LIN {X 0,Y 187.347,Z 253.939,A -85,B 0,C 180,E1 -26155.616,E2 -26155.616} C_VEL
LIN {X 0,Y 193.474,Z 262.012,A -85,B 0,C 180,E1 -26158.88,E2 -26158.88} C_VEL
LIN {X 0,Y 201.659,Z 270.756,A -85,B 0,C 180,E1 -26162.734,E2 -26162.734} C_VEL
LIN {X 0,Y 208.52,Z 276.532,A -85,B 0,C 180,E1 -26165.504,E2 -26165.504} C_VEL
LIN {X 0,Y 219.741,Z 283.992,A -85,B 0,C 180,E1 -26169.402,E2 -26169.402} C_VEL
LIN {X 0,Y 231.619,Z 290.129,A -85,B 0,C 180,E1 -26172.899,E2 -26172.899} C_VEL
LIN {X 0,Y 242.77,Z 294.984,A -85,B 0,C 180,E1 -26175.879,E2 -26175.879} C_VEL
LIN {X 0,Y 253.839,Z 299.442,A -85,B 0,C 180,E1 -26178.825,E2 -26178.825} C_VEL
LIN {X 0,Y 260.121,Z 302.011,A -85,B 0,C 180,E1 -26180.671,E2 -26180.671} C_VEL
LIN {X 0,Y 265.393,Z 304.118,A -85,B 0,C 180,E1 -26182.391,E2 -26182.391} C_VEL
LIN {X 0,Y 269.414,Z 305.803,A -85,B 0,C 180,E1 -26184.011,E2 -26184.011} C_VEL
LIN {X 0,Y 272.285,Z 307.103,A -85,B 0,C 180,E1 -26185.559,E2 -26185.559} C_VEL
LIN {X 0,Y 274.929,Z 308.026,A -85,B 0,C 180,E1 -26187.069,E2 -26187.069} C_VEL
LIN {X 0,Y 276.549,Z 308.577,A -85,B 0,C 180,E1 -26188.544,E2 -26188.544} C_VEL
LIN {X 0,Y 277.403,Z 308.756,A -85,B 0,C 180,E1 -26190,E2 -26190} C_VEL
LIN {X 0,Y 276.553,Z 308.577,A -85,B 0,C 180,E1 -26191.456,E2 -26191.456} C_VEL
LIN {X 0,Y 274.508,Z 307.901,A -85,B 0,C 180,E1 -26193.171,E2 -26193.171} C_VEL
LIN {X 0,Y 272.281,Z 307.103,A -85,B 0,C 180,E1 -26194.441,E2 -26194.441} C_VEL
LIN {X 0,Y 268.688,Z 305.506,A -85,B 0,C 180,E1 -26196.312,E2 -26196.312} C_VEL
LIN {X 0,Y 265.387,Z 304.118,A -85,B 0,C 180,E1 -26197.609,E2 -26197.609} C_VEL
LIN {X 0,Y 260.12,Z 302.01,A -85,B 0,C 180,E1 -26199.329,E2 -26199.329} C_VEL
LIN {X 0,Y 253.786,Z 299.444,A -85,B 0,C 180,E1 -26201.177,E2 -26201.177} C_VEL
LIN {X 0,Y 242.762,Z 295.002,A -85,B 0,C 180,E1 -26204.114,E2 -26204.114} C_VEL
LIN {X 0,Y 228.839,Z 288.795,A -85,B 0,C 180,E1 -26207.885,E2 -26207.885} C_VEL
LIN {X 0,Y 218.36,Z 283.205,A -85,B 0,C 180,E1 -26211.036,E2 -26211.036} C_VEL
LIN {X 0,Y 208.502,Z 276.573,A -85,B 0,C 180,E1 -26214.485,E2 -26214.485} C_VEL
LIN {X 0,Y 199.46,Z 268.628,A -85,B 0,C 180,E1 -26218.254,E2 -26218.254} C_VEL
LIN {X 0,Y 190.254,Z 257.902,A -85,B 0,C 180,E1 -26222.823,E2 -26222.823} C_VEL
LIN {X 0,Y 183.695,Z 248.177,A -85,B 0,C 180,E1 -26226.542,E2 -26226.542} C_VEL
LIN {X 0,Y 179.378,Z 240.181,A -85,B 0,C 180,E1 -26229.305,E2 -26229.305} C_VEL
LIN {X 0,Y 174.422,Z 229.195,A -85,B 0,C 180,E1 -26232.665,E2 -26232.665} C_VEL
LIN {X 0,Y 170.348,Z 218.871,A -85,B 0,C 180,E1 -26235.465,E2 -26235.465} C_VEL
LIN {X 0,Y 166.416,Z 207.712,A -85,B 0,C 180,E1 -26238.106,E2 -26238.106} C_VEL
LIN {X 0,Y 160.97,Z 191.989,A -85,B 0,C 180,E1 -26241.487,E2 -26241.487} C_VEL
LIN {X 0,Y 157.371,Z 183.213,A -85,B 0,C 180,E1 -26243.839,E2 -26243.839} C_VEL
LIN {X 0,Y 153.272,Z 174.648,A -85,B 0,C 180,E1 -26246.72,E2 -26246.72} C_VEL
LIN {X 0,Y 148.41,Z 165.755,A -85,B 0,C 180,E1 -26250.575,E2 -26250.575} C_VEL
LIN {X 0,Y 144.141,Z 158.771,A -85,B 0,C 180,E1 -26254.555,E2 -26254.555} C_VEL
LIN {X 0,Y 141.444,Z 154.774,A -85,B 0,C 180,E1 -26257.498,E2 -26257.498} C_VEL
LIN {X 0,Y 138.938,Z 150.996,A -85,B 0,C 180,E1 -26260.746,E2 -26260.746} C_VEL
LIN {X 0,Y 136.456,Z 147.585,A -85,B 0,C 180,E1 -26264.697,E2 -26264.697} C_VEL
LIN {X 0,Y 135.796,Z 146.33,A -85,B 0,C 180,E1 -26266.035,E2 -26266.035} C_VEL
LIN {X 0,Y 133.402,Z 143.471,A -85,B 0,C 180,E1 -26272.243,E2 -26272.243} C_VEL
LIN {X 0,Y 132.743,Z 141.518,A -85,B 0,C 180,E1 -26276.207,E2 -26276.207} C_VEL
LIN {X 0,Y 132.555,Z 140.915,A -85,B 0,C 180,E1 -26280.002,E2 -26280.002} C_VEL
LIN {X 0,Y 132.834,Z 141.773,A -85,B 0,C 180,E1 -26284.174,E2 -26284.174} C_VEL
LIN {X 0,Y 135.273,Z 145.963,A -85,B 0,C 180,E1 -26292.567,E2 -26292.567} C_VEL
LIN {X 0,Y 136.019,Z 146.575,A -85,B 0,C 180,E1 -26294.018,E2 -26294.018} C_VEL
LIN {X 0,Y 138.273,Z 150.297,A -85,B 0,C 180,E1 -26297.949,E2 -26297.949} C_VEL
LIN {X 0,Y 139.397,Z 151.65,A -85,B 0,C 180,E1 -26299.514,E2 -26299.514} C_VEL
LIN {X 0,Y 142.582,Z 156.425,A -85,B 0,C 180,E1 -26303.418,E2 -26303.418} C_VEL
LIN {X 0,Y 145.517,Z 161.05,A -85,B 0,C 180,E1 -26306.44,E2 -26306.44} C_VEL
LIN {X 0,Y 147.849,Z 164.954,A -85,B 0,C 180,E1 -26308.577,E2 -26308.577} C_VEL
LIN {X 0,Y 151.514,Z 173.302,A -85,B 0,C 180,E1 -26311.749,E2 -26311.749} C_VEL
LIN {X 0,Y 155.214,Z 183.268,A -85,B 0,C 180,E1 -26314.676,E2 -26314.676} C_VEL
LIN {X 0,Y 156.563,Z 187.492,A -85,B 0,C 180,E1 -26315.703,E2 -26315.703} C_VEL
LIN {X 0,Y 154.13,Z 215.499,A -85,B 0,C 180,E1 -26316.785,E2 -26316.785} C_VEL
LIN {X 0,Y 152.014,Z 228.263,A -85,B 0,C 180,E1 -26317.567,E2 -26317.567} C_VEL
LIN {X 0,Y 148.714,Z 241.034,A -85,B 0,C 180,E1 -26318.761,E2 -26318.761} C_VEL
LIN {X 0,Y 145.534,Z 250.542,A -85,B 0,C 180,E1 -26319.949,E2 -26319.949} C_VEL
LIN {X 0,Y 141.891,Z 259.814,A -85,B 0,C 180,E1 -26321.483,E2 -26321.483} C_VEL
LIN {X 0,Y 137.763,Z 268.752,A -85,B 0,C 180,E1 -26323.368,E2 -26323.368} C_VEL
LIN {X 0,Y 133.256,Z 277.274,A -85,B 0,C 180,E1 -26325.668,E2 -26325.668} C_VEL
LIN {X 0,Y 129.044,Z 284.489,A -85,B 0,C 180,E1 -26328.152,E2 -26328.152} C_VEL
LIN {X 0,Y 125.059,Z 290.686,A -85,B 0,C 180,E1 -26330.786,E2 -26330.786} C_VEL
LIN {X 0,Y 120.616,Z 297.224,A -85,B 0,C 180,E1 -26334.361,E2 -26334.361} C_VEL
LIN {X 0,Y 115.966,Z 303.643,A -85,B 0,C 180,E1 -26338.994,E2 -26338.994} C_VEL
LIN {X 0,Y 111.959,Z 308.773,A -85,B 0,C 180,E1 -26343.934,E2 -26343.934} C_VEL
LIN {X 0,Y 108.778,Z 312.762,A -85,B 0,C 180,E1 -26349.185,E2 -26349.185} C_VEL
LIN {X 0,Y 106.69,Z 315.721,A -85,B 0,C 180,E1 -26354.723,E2 -26354.723} C_VEL
LIN {X 0,Y 105.26,Z 318.183,A -85,B 0,C 180,E1 -26362.326,E2 -26362.326} C_VEL
LIN {X 0,Y 105.046,Z 318.779,A -85,B 0,C 180,E1 -26366.164,E2 -26366.164} C_VEL
LIN {X 0,Y 105.171,Z 318.941,A -85,B 0,C 180,E1 -26370,E2 -26370} C_VEL
LIN {X 0,Y 105.039,Z 318.779,A -85,B 0,C 180,E1 -26373.836,E2 -26373.836} C_VEL
LIN {X 0,Y 105.229,Z 318.182,A -85,B 0,C 180,E1 -26377.676,E2 -26377.676} C_VEL
LIN {X 0,Y 106.69,Z 315.721,A -85,B 0,C 180,E1 -26385.277,E2 -26385.277} C_VEL
LIN {X 0,Y 108.778,Z 312.762,A -85,B 0,C 180,E1 -26390.815,E2 -26390.815} C_VEL
LIN {X 0,Y 111.96,Z 308.773,A -85,B 0,C 180,E1 -26396.066,E2 -26396.066} C_VEL
LIN {X 0,Y 115.976,Z 303.644,A -85,B 0,C 180,E1 -26401.003,E2 -26401.003} C_VEL
LIN {X 0,Y 120.658,Z 297.225,A -85,B 0,C 180,E1 -26405.625,E2 -26405.625} C_VEL
LIN {X 0,Y 126.044,Z 289.304,A -85,B 0,C 180,E1 -26409.883,E2 -26409.883} C_VEL
LIN {X 0,Y 131.143,Z 281.111,A -85,B 0,C 180,E1 -26413.1,E2 -26413.1} C_VEL
LIN {X 0,Y 136.058,Z 272.154,A -85,B 0,C 180,E1 -26415.783,E2 -26415.783} C_VEL
LIN {X 0,Y 140.108,Z 263.865,A -85,B 0,C 180,E1 -26417.721,E2 -26417.721} C_VEL
LIN {X 0,Y 144.302,Z 253.804,A -85,B 0,C 180,E1 -26419.552,E2 -26419.552} C_VEL
LIN {X 0,Y 147.751,Z 244.053,A -85,B 0,C 180,E1 -26420.889,E2 -26420.889} C_VEL
LIN {X 0,Y 150.612,Z 233.975,A -85,B 0,C 180,E1 -26421.947,E2 -26421.947} C_VEL
LIN {X 0,Y 152.841,Z 223.594,A -85,B 0,C 180,E1 -26422.756,E2 -26422.756} C_VEL
LIN {X 0,Y 154.336,Z 213.507,A -85,B 0,C 180,E1 -26423.307,E2 -26423.307} C_VEL
LIN {X 0,Y 156.557,Z 187.548,A -85,B 0,C 180,E1 -26424.295,E2 -26424.295} C_VEL
LIN {X 0,Y 153.767,Z 179.164,A -85,B 0,C 180,E1 -26426.442,E2 -26426.442} C_VEL
LIN {X 0,Y 149.574,Z 168.715,A -85,B 0,C 180,E1 -26429.888,E2 -26429.888} C_VEL
LIN {X 0,Y 146.975,Z 163.379,A -85,B 0,C 180,E1 -26432.209,E2 -26432.209} C_VEL
LIN {X 0,Y 143.653,Z 158.1,A -85,B 0,C 180,E1 -26435.426,E2 -26435.426} C_VEL
LIN {X 0,Y 141.524,Z 154.839,A -85,B 0,C 180,E1 -26437.787,E2 -26437.787} C_VEL
LIN {X 0,Y 138.836,Z 150.858,A -85,B 0,C 180,E1 -26441.267,E2 -26441.267} C_VEL
LIN {X 0,Y 138.374,Z 150.375,A -85,B 0,C 180,E1 -26441.912,E2 -26441.912} C_VEL
LIN {X 0,Y 136.784,Z 149.34,A -85,B 0,C 180,E1 -26444.241,E2 -26444.241} C_VEL
LIN {X 0,Y 134.384,Z 149.472,A -85,B 0,C 180,E1 -26448.305,E2 -26448.305} C_VEL
LIN {X 0,Y 132.917,Z 149.898,A -85,B 0,C 180,E1 -26451.671,E2 -26451.671} C_VEL
LIN {X 0,Y 132.203,Z 149.602,A -85,B 0,C 180,E1 -26454.227,E2 -26454.227} C_VEL
LIN {X 0,Y 132.052,Z 149.284,A -85,B 0,C 180,E1 -26455.075,E2 -26455.075} C_VEL
LIN {X 0,Y 131.771,Z 148.3,A -85,B 0,C 180,E1 -26457.706,E2 -26457.706} C_VEL
LIN {X 0,Y 131.686,Z 147.992,A -85,B 0,C 180,E1 -26459.998,E2 -26459.998} C_VEL
LIN {X 0,Y 131.916,Z 148.746,A -85,B 0,C 180,E1 -26464.199,E2 -26464.199} C_VEL
LIN {X 0,Y 133.989,Z 152.766,A -85,B 0,C 180,E1 -26472.109,E2 -26472.109} C_VEL
LIN {X 0,Y 134.836,Z 153.712,A -85,B 0,C 180,E1 -26473.919,E2 -26473.919} C_VEL
LIN {X 0,Y 137.218,Z 157.472,A -85,B 0,C 180,E1 -26478.163,E2 -26478.163} C_VEL
LIN {X 0,Y 140.448,Z 162.453,A -85,B 0,C 180,E1 -26482.525,E2 -26482.525} C_VEL
LIN {X 0,Y 143.306,Z 167.161,A -85,B 0,C 180,E1 -26485.702,E2 -26485.702} C_VEL
LIN {X 0,Y 146.753,Z 173.26,A -85,B 0,C 180,E1 -26489.003,E2 -26489.003} C_VEL
LIN {X 0,Y 151.229,Z 182.072,A -85,B 0,C 180,E1 -26492.72,E2 -26492.72} C_VEL
LIN {X 0,Y 155.275,Z 191.24,A -85,B 0,C 180,E1 -26495.712,E2 -26495.712} C_VEL
LIN {X 0,Y 159.125,Z 202.11,A -85,B 0,C 180,E1 -26498.394,E2 -26498.394} C_VEL
LIN {X 0,Y 163.336,Z 215.721,A -85,B 0,C 180,E1 -26501.519,E2 -26501.519} C_VEL
LIN {X 0,Y 166.6,Z 225.797,A -85,B 0,C 180,E1 -26504.181,E2 -26504.181} C_VEL
LIN {X 0,Y 170.345,Z 235.871,A -85,B 0,C 180,E1 -26507.235,E2 -26507.235} C_VEL
LIN {X 0,Y 174.011,Z 244.448,A -85,B 0,C 180,E1 -26510.117,E2 -26510.117} C_VEL
LIN {X 0,Y 178.938,Z 253.723,A -85,B 0,C 180,E1 -26513.626,E2 -26513.626} C_VEL
LIN {X 0,Y 184.314,Z 261.859,A -85,B 0,C 180,E1 -26517.019,E2 -26517.019} C_VEL
LIN {X 0,Y 190.756,Z 269.605,A -85,B 0,C 180,E1 -26520.561,E2 -26520.561} C_VEL
LIN {X 0,Y 198.398,Z 276.897,A -85,B 0,C 180,E1 -26524.191,E2 -26524.191} C_VEL
LIN {X 0,Y 208.728,Z 284.302,A -85,B 0,C 180,E1 -26528.261,E2 -26528.261} C_VEL
LIN {X 0,Y 221.275,Z 291.024,A -85,B 0,C 180,E1 -26532.33,E2 -26532.33} C_VEL
LIN {X 0,Y 235.088,Z 296.772,A -85,B 0,C 180,E1 -26536.163,E2 -26536.163} C_VEL
LIN {X 0,Y 246.761,Z 301.009,A -85,B 0,C 180,E1 -26539.289,E2 -26539.289} C_VEL
LIN {X 0,Y 255.566,Z 304.111,A -85,B 0,C 180,E1 -26541.88,E2 -26541.88} C_VEL
LIN {X 0,Y 261.468,Z 306.181,A -85,B 0,C 180,E1 -26543.991,E2 -26543.991} C_VEL
LIN {X 0,Y 264.422,Z 307.313,A -85,B 0,C 180,E1 -26545.427,E2 -26545.427} C_VEL
LIN {X 0,Y 267.407,Z 308.28,A -85,B 0,C 180,E1 -26547.077,E2 -26547.077} C_VEL
LIN {X 0,Y 269.225,Z 308.773,A -85,B 0,C 180,E1 -26548.504,E2 -26548.504} C_VEL
LIN {X 0,Y 270.244,Z 308.944,A -85,B 0,C 180,E1 -26550,E2 -26550} C_VEL
LIN {X 0,Y 269.227,Z 308.772,A -85,B 0,C 180,E1 -26551.496,E2 -26551.496} C_VEL
LIN {X 0,Y 267.241,Z 308.234,A -85,B 0,C 180,E1 -26553.015,E2 -26553.015} C_VEL
LIN {X 0,Y 264.419,Z 307.313,A -85,B 0,C 180,E1 -26554.573,E2 -26554.573} C_VEL
LIN {X 0,Y 261.017,Z 306.031,A -85,B 0,C 180,E1 -26556.183,E2 -26556.183} C_VEL
LIN {X 0,Y 255.566,Z 304.112,A -85,B 0,C 180,E1 -26558.12,E2 -26558.12} C_VEL
LIN {X 0,Y 249.675,Z 302.059,A -85,B 0,C 180,E1 -26559.875,E2 -26559.875} C_VEL
LIN {X 0,Y 243.086,Z 299.734,A -85,B 0,C 180,E1 -26561.676,E2 -26561.676} C_VEL
LIN {X 0,Y 232.334,Z 295.749,A -85,B 0,C 180,E1 -26564.541,E2 -26564.541} C_VEL
LIN {X 0,Y 221.274,Z 291.028,A -85,B 0,C 180,E1 -26567.669,E2 -26567.669} C_VEL
LIN {X 0,Y 208.718,Z 284.302,A -85,B 0,C 180,E1 -26571.74,E2 -26571.74} C_VEL
LIN {X 0,Y 200.627,Z 278.691,A -85,B 0,C 180,E1 -26574.857,E2 -26574.857} C_VEL
LIN {X 0,Y 192.263,Z 271.143,A -85,B 0,C 180,E1 -26578.684,E2 -26578.684} C_VEL
LIN {X 0,Y 185.27,Z 263.055,A -85,B 0,C 180,E1 -26582.435,E2 -26582.435} C_VEL
LIN {X 0,Y 179.577,Z 254.766,A -85,B 0,C 180,E1 -26585.947,E2 -26585.947} C_VEL
LIN {X 0,Y 174.772,Z 246.129,A -85,B 0,C 180,E1 -26589.28,E2 -26589.28} C_VEL
LIN {X 0,Y 170.953,Z 237.377,A -85,B 0,C 180,E1 -26592.271,E2 -26592.271} C_VEL
LIN {X 0,Y 168.007,Z 229.673,A -85,B 0,C 180,E1 -26594.674,E2 -26594.674} C_VEL
LIN {X 0,Y 164.616,Z 219.813,A -85,B 0,C 180,E1 -26597.437,E2 -26597.437} C_VEL
LIN {X 0,Y 161.141,Z 208.708,A -85,B 0,C 180,E1 -26600.167,E2 -26600.167} C_VEL
LIN {X 0,Y 156.949,Z 195.782,A -85,B 0,C 180,E1 -26603.099,E2 -26603.099} C_VEL
LIN {X 0,Y 153.641,Z 187.418,A -85,B 0,C 180,E1 -26605.46,E2 -26605.46} C_VEL
LIN {X 0,Y 149.751,Z 179.066,A -85,B 0,C 180,E1 -26608.448,E2 -26608.448} C_VEL
LIN {X 0,Y 145.615,Z 171.171,A -85,B 0,C 180,E1 -26612.038,E2 -26612.038} C_VEL
LIN {X 0,Y 142.066,Z 165.032,A -85,B 0,C 180,E1 -26615.623,E2 -26615.623} C_VEL
LIN {X 0,Y 139.445,Z 160.96,A -85,B 0,C 180,E1 -26618.708,E2 -26618.708} C_VEL
LIN {X 0,Y 137.219,Z 157.462,A -85,B 0,C 180,E1 -26621.838,E2 -26621.838} C_VEL
LIN {X 0,Y 134.845,Z 153.736,A -85,B 0,C 180,E1 -26626.06,E2 -26626.06} C_VEL
LIN {X 0,Y 134.213,Z 152.941,A -85,B 0,C 180,E1 -26627.402,E2 -26627.402} C_VEL
LIN {X 0,Y 132.168,Z 149.79,A -85,B 0,C 180,E1 -26633.897,E2 -26633.897} C_VEL
LIN {X 0,Y 131.802,Z 148.388,A -85,B 0,C 180,E1 -26636.945,E2 -26636.945} C_VEL
LIN {X 0,Y 131.689,Z 147.971,A -85,B 0,C 180,E1 -26640.002,E2 -26640.002} C_VEL
LIN {X 0,Y 131.92,Z 148.834,A -85,B 0,C 180,E1 -26643.916,E2 -26643.916} C_VEL
LIN {X 0,Y 134.157,Z 152.888,A -85,B 0,C 180,E1 -26652.097,E2 -26652.097} C_VEL
LIN {X 0,Y 134.767,Z 153.539,A -85,B 0,C 180,E1 -26653.382,E2 -26653.382} C_VEL
LIN {X 0,Y 137.292,Z 157.526,A -85,B 0,C 180,E1 -26657.889,E2 -26657.889} C_VEL
LIN {X 0,Y 140.634,Z 162.769,A -85,B 0,C 180,E1 -26662.373,E2 -26662.373} C_VEL
LIN {X 0,Y 144.114,Z 168.46,A -85,B 0,C 180,E1 -26666.133,E2 -26666.133} C_VEL
LIN {X 0,Y 146.33,Z 173.167,A -85,B 0,C 180,E1 -26668.314,E2 -26668.314} C_VEL
LIN {X 0,Y 149.507,Z 181.45,A -85,B 0,C 180,E1 -26671.237,E2 -26671.237} C_VEL
LIN {X 0,Y 151.852,Z 188.359,A -85,B 0,C 180,E1 -26673.242,E2 -26673.242} C_VEL
LIN {X 0,Y 152.309,Z 189.835,A -85,B 0,C 180,E1 -26673.624,E2 -26673.624} C_VEL
LIN {X 0,Y 150.029,Z 215.003,A -85,B 0,C 180,E1 -26674.599,E2 -26674.599} C_VEL
LIN {X 0,Y 147.671,Z 228.649,A -85,B 0,C 180,E1 -26675.428,E2 -26675.428} C_VEL
LIN {X 0,Y 144.38,Z 240.843,A -85,B 0,C 180,E1 -26676.566,E2 -26676.566} C_VEL
LIN {X 0,Y 141.084,Z 250.352,A -85,B 0,C 180,E1 -26677.74,E2 -26677.74} C_VEL
LIN {X 0,Y 137.277,Z 259.622,A -85,B 0,C 180,E1 -26679.255,E2 -26679.255} C_VEL
LIN {X 0,Y 132.98,Z 268.562,A -85,B 0,C 180,E1 -26681.139,E2 -26681.139} C_VEL
LIN {X 0,Y 128.274,Z 277.084,A -85,B 0,C 180,E1 -26683.452,E2 -26683.452} C_VEL
LIN {X 0,Y 123.816,Z 284.298,A -85,B 0,C 180,E1 -26685.947,E2 -26685.947} C_VEL
LIN {X 0,Y 119.631,Z 290.495,A -85,B 0,C 180,E1 -26688.631,E2 -26688.631} C_VEL
LIN {X 0,Y 114.885,Z 297.032,A -85,B 0,C 180,E1 -26692.284,E2 -26692.284} C_VEL
LIN {X 0,Y 109.928,Z 303.453,A -85,B 0,C 180,E1 -26697.083,E2 -26697.083} C_VEL
LIN {X 0,Y 105.593,Z 308.581,A -85,B 0,C 180,E1 -26702.231,E2 -26702.231} C_VEL
LIN {X 0,Y 102.159,Z 312.571,A -85,B 0,C 180,E1 -26707.767,E2 -26707.767} C_VEL
LIN {X 0,Y 99.814,Z 315.529,A -85,B 0,C 180,E1 -26713.642,E2 -26713.642} C_VEL
LIN {X 0,Y 98.209,Z 317.992,A -85,B 0,C 180,E1 -26721.771,E2 -26721.771} C_VEL
LIN {X 0,Y 97.952,Z 318.588,A -85,B 0,C 180,E1 -26725.886,E2 -26725.886} C_VEL
LIN {X 0,Y 98.077,Z 318.75,A -85,B 0,C 180,E1 -26730,E2 -26730} C_VEL
LIN {X 0,Y 97.945,Z 318.588,A -85,B 0,C 180,E1 -26734.115,E2 -26734.115} C_VEL
LIN {X 0,Y 98.185,Z 317.991,A -85,B 0,C 180,E1 -26738.231,E2 -26738.231} C_VEL
LIN {X 0,Y 99.813,Z 315.529,A -85,B 0,C 180,E1 -26746.358,E2 -26746.358} C_VEL
LIN {X 0,Y 102.159,Z 312.571,A -85,B 0,C 180,E1 -26752.233,E2 -26752.233} C_VEL
LIN {X 0,Y 105.594,Z 308.581,A -85,B 0,C 180,E1 -26757.768,E2 -26757.768} C_VEL
LIN {X 0,Y 109.938,Z 303.453,A -85,B 0,C 180,E1 -26762.914,E2 -26762.914} C_VEL
LIN {X 0,Y 114.094,Z 298.136,A -85,B 0,C 180,E1 -26766.962,E2 -26766.962} C_VEL
LIN {X 0,Y 118.659,Z 291.872,A -85,B 0,C 180,E1 -26770.656,E2 -26770.656} C_VEL
LIN {X 0,Y 122.786,Z 285.925,A -85,B 0,C 180,E1 -26773.381,E2 -26773.381} C_VEL
LIN {X 0,Y 127.158,Z 279.002,A -85,B 0,C 180,E1 -26775.931,E2 -26775.931} C_VEL
LIN {X 0,Y 131.793,Z 270.829,A -85,B 0,C 180,E1 -26778.293,E2 -26778.293} C_VEL
LIN {X 0,Y 136.04,Z 262.324,A -85,B 0,C 180,E1 -26780.216,E2 -26780.216} C_VEL
LIN {X 0,Y 139.797,Z 253.614,A -85,B 0,C 180,E1 -26781.768,E2 -26781.768} C_VEL
LIN {X 0,Y 143.385,Z 243.862,A -85,B 0,C 180,E1 -26783.087,E2 -26783.087} C_VEL
LIN {X 0,Y 146.345,Z 233.785,A -85,B 0,C 180,E1 -26784.134,E2 -26784.134} C_VEL
LIN {X 0,Y 148.503,Z 224.159,A -85,B 0,C 180,E1 -26784.888,E2 -26784.888} C_VEL
LIN {X 0,Y 150.129,Z 214.001,A -85,B 0,C 180,E1 -26785.444,E2 -26785.444} C_VEL
LIN {X 0,Y 152.308,Z 189.849,A -85,B 0,C 180,E1 -26786.376,E2 -26786.376} C_VEL
LIN {X 0,Y 149.428,Z 181.119,A -85,B 0,C 180,E1 -26788.843,E2 -26788.843} C_VEL
LIN {X 0,Y 145.916,Z 172.188,A -85,B 0,C 180,E1 -26792.087,E2 -26792.087} C_VEL
LIN {X 0,Y 143.864,Z 168.091,A -85,B 0,C 180,E1 -26794.11,E2 -26794.11} C_VEL
LIN {X 0,Y 140.03,Z 161.67,A -85,B 0,C 180,E1 -26798.378,E2 -26798.378} C_VEL
LIN {X 0,Y 137.175,Z 157.365,A -85,B 0,C 180,E1 -26802.288,E2 -26802.288} C_VEL
LIN {X 0,Y 134.848,Z 153.726,A -85,B 0,C 180,E1 -26806.434,E2 -26806.434} C_VEL
LIN {X 0,Y 133.988,Z 152.722,A -85,B 0,C 180,E1 -26808.28,E2 -26808.28} C_VEL
LIN {X 0,Y 132.052,Z 149.284,A -85,B 0,C 180,E1 -26815.075,E2 -26815.075} C_VEL
LIN {X 0,Y 131.795,Z 149.015,A -85,B 0,C 180,E1 -26816.766,E2 -26816.766} C_VEL
LIN {X 0,Y 131.555,Z 149.546,A -85,B 0,C 180,E1 -26818.456,E2 -26818.456} C_VEL
LIN {X 0,Y 131.226,Z 152.124,A -85,B 0,C 180,E1 -26821.743,E2 -26821.743} C_VEL
LIN {X 0,Y 131.419,Z 157.072,A -85,B 0,C 180,E1 -26826.703,E2 -26826.703} C_VEL
LIN {X 0,Y 131.788,Z 158.208,A -85,B 0,C 180,E1 -26828.417,E2 -26828.417} C_VEL
LIN {X 0,Y 133.501,Z 160.371,A -85,B 0,C 180,E1 -26833.024,E2 -26833.024} C_VEL
LIN {X 0,Y 135.841,Z 164.254,A -85,B 0,C 180,E1 -26837.499,E2 -26837.499} C_VEL
LIN {X 0,Y 138.745,Z 169.153,A -85,B 0,C 180,E1 -26841.693,E2 -26841.693} C_VEL
LIN {X 0,Y 141.976,Z 174.705,A -85,B 0,C 180,E1 -26845.444,E2 -26845.444} C_VEL
LIN {X 0,Y 145.7,Z 182.086,A -85,B 0,C 180,E1 -26849.134,E2 -26849.134} C_VEL
LIN {X 0,Y 149.653,Z 190.686,A -85,B 0,C 180,E1 -26852.526,E2 -26852.526} C_VEL
LIN {X 0,Y 152.731,Z 198.624,A -85,B 0,C 180,E1 -26854.953,E2 -26854.953} C_VEL
LIN {X 0,Y 155.703,Z 208.241,A -85,B 0,C 180,E1 -26857.337,E2 -26857.337} C_VEL
LIN {X 0,Y 158.276,Z 217.717,A -85,B 0,C 180,E1 -26859.663,E2 -26859.663} C_VEL
LIN {X 0,Y 160.592,Z 226.033,A -85,B 0,C 180,E1 -26861.929,E2 -26861.929} C_VEL
LIN {X 0,Y 163.82,Z 236.323,A -85,B 0,C 180,E1 -26865.134,E2 -26865.134} C_VEL
LIN {X 0,Y 167.078,Z 245.062,A -85,B 0,C 180,E1 -26868.195,E2 -26868.195} C_VEL
LIN {X 0,Y 170.806,Z 253.395,A -85,B 0,C 180,E1 -26871.421,E2 -26871.421} C_VEL
LIN {X 0,Y 176.31,Z 262.848,A -85,B 0,C 180,E1 -26875.544,E2 -26875.544} C_VEL
LIN {X 0,Y 181.672,Z 269.902,A -85,B 0,C 180,E1 -26878.939,E2 -26878.939} C_VEL
LIN {X 0,Y 189.208,Z 277.748,A -85,B 0,C 180,E1 -26883.055,E2 -26883.055} C_VEL
LIN {X 0,Y 196.205,Z 283.309,A -85,B 0,C 180,E1 -26886.237,E2 -26886.237} C_VEL
LIN {X 0,Y 206.126,Z 289.433,A -85,B 0,C 180,E1 -26890.065,E2 -26890.065} C_VEL
LIN {X 0,Y 214.695,Z 293.589,A -85,B 0,C 180,E1 -26892.866,E2 -26892.866} C_VEL
LIN {X 0,Y 224.751,Z 297.544,A -85,B 0,C 180,E1 -26895.779,E2 -26895.779} C_VEL
LIN {X 0,Y 236.33,Z 301.449,A -85,B 0,C 180,E1 -26898.913,E2 -26898.913} C_VEL
LIN {X 0,Y 242.253,Z 303.263,A -85,B 0,C 180,E1 -26900.524,E2 -26900.524} C_VEL
LIN {X 0,Y 248.217,Z 305.083,A -85,B 0,C 180,E1 -26902.295,E2 -26902.295} C_VEL
LIN {X 0,Y 254.241,Z 306.884,A -85,B 0,C 180,E1 -26904.345,E2 -26904.345} C_VEL
LIN {X 0,Y 256.353,Z 307.528,A -85,B 0,C 180,E1 -26905.282,E2 -26905.282} C_VEL
LIN {X 0,Y 260.307,Z 308.642,A -85,B 0,C 180,E1 -26907.363,E2 -26907.363} C_VEL
LIN {X 0,Y 261.81,Z 308.971,A -85,B 0,C 180,E1 -26908.462,E2 -26908.462} C_VEL
LIN {X 0,Y 263.065,Z 309.133,A -85,B 0,C 180,E1 -26910,E2 -26910} C_VEL
LIN {X 0,Y 261.811,Z 308.971,A -85,B 0,C 180,E1 -26911.538,E2 -26911.538} C_VEL
LIN {X 0,Y 259.439,Z 308.445,A -85,B 0,C 180,E1 -26913.106,E2 -26913.106} C_VEL
LIN {X 0,Y 256.337,Z 307.529,A -85,B 0,C 180,E1 -26914.718,E2 -26914.718} C_VEL
LIN {X 0,Y 254.241,Z 306.885,A -85,B 0,C 180,E1 -26915.654,E2 -26915.654} C_VEL
LIN {X 0,Y 248.216,Z 305.083,A -85,B 0,C 180,E1 -26917.705,E2 -26917.705} C_VEL
LIN {X 0,Y 239.845,Z 302.553,A -85,B 0,C 180,E1 -26920.126,E2 -26920.126} C_VEL
LIN {X 0,Y 230.48,Z 299.542,A -85,B 0,C 180,E1 -26922.643,E2 -26922.643} C_VEL
LIN {X 0,Y 219.124,Z 295.381,A -85,B 0,C 180,E1 -26925.809,E2 -26925.809} C_VEL
LIN {X 0,Y 208.33,Z 290.583,A -85,B 0,C 180,E1 -26929.168,E2 -26929.168} C_VEL
LIN {X 0,Y 198.008,Z 284.605,A -85,B 0,C 180,E1 -26932.981,E2 -26932.981} C_VEL
LIN {X 0,Y 189.203,Z 277.758,A -85,B 0,C 180,E1 -26936.942,E2 -26936.942} C_VEL
LIN {X 0,Y 181.143,Z 269.224,A -85,B 0,C 180,E1 -26941.402,E2 -26941.402} C_VEL
LIN {X 0,Y 174.04,Z 259.139,A -85,B 0,C 180,E1 -26946.137,E2 -26946.137} C_VEL
LIN {X 0,Y 169.101,Z 249.83,A -85,B 0,C 180,E1 -26950.016,E2 -26950.016} C_VEL
LIN {X 0,Y 165.101,Z 239.932,A -85,B 0,C 180,E1 -26953.645,E2 -26953.645} C_VEL
LIN {X 0,Y 162.009,Z 230.667,A -85,B 0,C 180,E1 -26956.675,E2 -26956.675} C_VEL
LIN {X 0,Y 158.932,Z 220.126,A -85,B 0,C 180,E1 -26959.707,E2 -26959.707} C_VEL
LIN {X 0,Y 156.105,Z 209.559,A -85,B 0,C 180,E1 -26962.369,E2 -26962.369} C_VEL
LIN {X 0,Y 152.73,Z 198.678,A -85,B 0,C 180,E1 -26965.043,E2 -26965.043} C_VEL
LIN {X 0,Y 149.485,Z 190.266,A -85,B 0,C 180,E1 -26967.612,E2 -26967.612} C_VEL
LIN {X 0,Y 145.277,Z 181.17,A -85,B 0,C 180,E1 -26971.262,E2 -26971.262} C_VEL
LIN {X 0,Y 141.682,Z 174.203,A -85,B 0,C 180,E1 -26974.868,E2 -26974.868} C_VEL
LIN {X 0,Y 138.126,Z 167.978,A -85,B 0,C 180,E1 -26979.137,E2 -26979.137} C_VEL
LIN {X 0,Y 135.64,Z 164.033,A -85,B 0,C 180,E1 -26982.814,E2 -26982.814} C_VEL
LIN {X 0,Y 133.36,Z 160.063,A -85,B 0,C 180,E1 -26987.32,E2 -26987.32} C_VEL
LIN {X 0,Y 131.236,Z 156.88,A -85,B 0,C 180,E1 -26994.142,E2 -26994.142} C_VEL
LIN {X 0,Y 130.876,Z 155.31,A -85,B 0,C 180,E1 -26997.693,E2 -26997.693} C_VEL
LIN {X 0,Y 130.822,Z 155.026,A -85,B 0,C 180,E1 -27000.002,E2 -27000.002} C_VEL
LIN {X 0,Y 130.987,Z 155.731,A -85,B 0,C 180,E1 -27003.366,E2 -27003.366} C_VEL
LIN {X 0,Y 133.135,Z 159.885,A -85,B 0,C 180,E1 -27011.813,E2 -27011.813} C_VEL
LIN {X 0,Y 133.673,Z 160.769,A -85,B 0,C 180,E1 -27013.058,E2 -27013.058} C_VEL
LIN {X 0,Y 136.276,Z 165.054,A -85,B 0,C 180,E1 -27017.832,E2 -27017.832} C_VEL
LIN {X 0,Y 138.79,Z 169.209,A -85,B 0,C 180,E1 -27021.37,E2 -27021.37} C_VEL
LIN {X 0,Y 141.981,Z 174.773,A -85,B 0,C 180,E1 -27025.079,E2 -27025.079} C_VEL
LIN {X 0,Y 144.304,Z 180.391,A -85,B 0,C 180,E1 -27027.561,E2 -27027.561} C_VEL
LIN {X 0,Y 147.873,Z 190.744,A -85,B 0,C 180,E1 -27031.048,E2 -27031.048} C_VEL
LIN {X 0,Y 148.276,Z 192.275,A -85,B 0,C 180,E1 -27031.443,E2 -27031.443} C_VEL
LIN {X 0,Y 146.023,Z 215.571,A -85,B 0,C 180,E1 -27032.346,E2 -27032.346} C_VEL
LIN {X 0,Y 143.399,Z 229.562,A -85,B 0,C 180,E1 -27033.213,E2 -27033.213} C_VEL
LIN {X 0,Y 140.263,Z 240.653,A -85,B 0,C 180,E1 -27034.234,E2 -27034.234} C_VEL
LIN {X 0,Y 136.861,Z 250.162,A -85,B 0,C 180,E1 -27035.393,E2 -27035.393} C_VEL
LIN {X 0,Y 132.905,Z 259.432,A -85,B 0,C 180,E1 -27036.889,E2 -27036.889} C_VEL
LIN {X 0,Y 128.422,Z 268.371,A -85,B 0,C 180,E1 -27038.754,E2 -27038.754} C_VEL
LIN {X 0,Y 123.485,Z 276.893,A -85,B 0,C 180,E1 -27041.053,E2 -27041.053} C_VEL
LIN {X 0,Y 118.799,Z 284.107,A -85,B 0,C 180,E1 -27043.557,E2 -27043.557} C_VEL
LIN {X 0,Y 114.378,Z 290.304,A -85,B 0,C 180,E1 -27046.27,E2 -27046.27} C_VEL
LIN {X 0,Y 109.324,Z 296.84,A -85,B 0,C 180,E1 -27049.995,E2 -27049.995} C_VEL
LIN {X 0,Y 105.7,Z 301.344,A -85,B 0,C 180,E1 -27053.244,E2 -27053.244} C_VEL
LIN {X 0,Y 100.749,Z 306.835,A -85,B 0,C 180,E1 -27058.454,E2 -27058.454} C_VEL
LIN {X 0,Y 96.741,Z 311.162,A -85,B 0,C 180,E1 -27064.158,E2 -27064.158} C_VEL
LIN {X 0,Y 94.561,Z 313.531,A -85,B 0,C 180,E1 -27068.185,E2 -27068.185} C_VEL
LIN {X 0,Y 92.987,Z 315.338,A -85,B 0,C 180,E1 -27072.403,E2 -27072.403} C_VEL
LIN {X 0,Y 91.163,Z 317.8,A -85,B 0,C 180,E1 -27081.13,E2 -27081.13} C_VEL
LIN {X 0,Y 90.88,Z 318.398,A -85,B 0,C 180,E1 -27085.565,E2 -27085.565} C_VEL
LIN {X 0,Y 90.976,Z 318.56,A -85,B 0,C 180,E1 -27090,E2 -27090} C_VEL
LIN {X 0,Y 90.874,Z 318.398,A -85,B 0,C 180,E1 -27094.436,E2 -27094.436} C_VEL
LIN {X 0,Y 91.145,Z 317.8,A -85,B 0,C 180,E1 -27098.871,E2 -27098.871} C_VEL
LIN {X 0,Y 92.987,Z 315.338,A -85,B 0,C 180,E1 -27107.597,E2 -27107.597} C_VEL
LIN {X 0,Y 95.587,Z 312.38,A -85,B 0,C 180,E1 -27113.853,E2 -27113.853} C_VEL
LIN {X 0,Y 99.322,Z 308.389,A -85,B 0,C 180,E1 -27119.691,E2 -27119.691} C_VEL
LIN {X 0,Y 104.016,Z 303.261,A -85,B 0,C 180,E1 -27125.052,E2 -27125.052} C_VEL
LIN {X 0,Y 109.366,Z 296.842,A -85,B 0,C 180,E1 -27129.987,E2 -27129.987} C_VEL
LIN {X 0,Y 115.494,Z 288.923,A -85,B 0,C 180,E1 -27134.41,E2 -27134.41} C_VEL
LIN {X 0,Y 121.145,Z 280.73,A -85,B 0,C 180,E1 -27137.703,E2 -27137.703} C_VEL
LIN {X 0,Y 126.564,Z 271.773,A -85,B 0,C 180,E1 -27140.396,E2 -27140.396} C_VEL
LIN {X 0,Y 130.963,Z 263.484,A -85,B 0,C 180,E1 -27142.33,E2 -27142.33} C_VEL
LIN {X 0,Y 135.519,Z 253.423,A -85,B 0,C 180,E1 -27144.126,E2 -27144.126} C_VEL
LIN {X 0,Y 139.247,Z 243.672,A -85,B 0,C 180,E1 -27145.418,E2 -27145.418} C_VEL
LIN {X 0,Y 142.309,Z 233.595,A -85,B 0,C 180,E1 -27146.447,E2 -27146.447} C_VEL
LIN {X 0,Y 144.663,Z 223.367,A -85,B 0,C 180,E1 -27147.224,E2 -27147.224} C_VEL
LIN {X 0,Y 146.319,Z 212.946,A -85,B 0,C 180,E1 -27147.778,E2 -27147.778} C_VEL
LIN {X 0,Y 148.203,Z 192.001,A -85,B 0,C 180,E1 -27148.628,E2 -27148.628} C_VEL
LIN {X 0,Y 145.262,Z 183.058,A -85,B 0,C 180,E1 -27151.459,E2 -27151.459} C_VEL
LIN {X 0,Y 142.596,Z 176.072,A -85,B 0,C 180,E1 -27154.256,E2 -27154.256} C_VEL
LIN {X 0,Y 139.717,Z 170.752,A -85,B 0,C 180,E1 -27157.485,E2 -27157.485} C_VEL
LIN {X 0,Y 137.591,Z 167.268,A -85,B 0,C 180,E1 -27160.219,E2 -27160.219} C_VEL
LIN {X 0,Y 135.503,Z 163.804,A -85,B 0,C 180,E1 -27163.424,E2 -27163.424} C_VEL
LIN {X 0,Y 133.303,Z 160.002,A -85,B 0,C 180,E1 -27167.824,E2 -27167.824} C_VEL
LIN {X 0,Y 131.166,Z 156.589,A -85,B 0,C 180,E1 -27175.003,E2 -27175.003} C_VEL
LIN {X 0,Y 130.902,Z 155.382,A -85,B 0,C 180,E1 -27177.691,E2 -27177.691} C_VEL
LIN {X 0,Y 130.821,Z 155.036,A -85,B 0,C 180,E1 -27179.998,E2 -27179.998} C_VEL
LIN {X 0,Y 130.998,Z 155.758,A -85,B 0,C 180,E1 -27183.844,E2 -27183.844} C_VEL
LIN {X 0,Y 131.788,Z 158.208,A -85,B 0,C 180,E1 -27188.417,E2 -27188.417} C_VEL
LIN {X 0,Y 132.467,Z 160.138,A -85,B 0,C 180,E1 -27190.818,E2 -27190.818} C_VEL
LIN {X 0,Y 133.167,Z 163.054,A -85,B 0,C 180,E1 -27193.031,E2 -27193.031} C_VEL
LIN {X 0,Y 134.825,Z 170.139,A -85,B 0,C 180,E1 -27197.142,E2 -27197.142} C_VEL
LIN {X 0,Y 136.438,Z 174.52,A -85,B 0,C 180,E1 -27199.918,E2 -27199.918} C_VEL
LIN {X 0,Y 139.695,Z 180.608,A -85,B 0,C 180,E1 -27204.125,E2 -27204.125} C_VEL
LIN {X 0,Y 143.392,Z 188.388,A -85,B 0,C 180,E1 -27208.089,E2 -27208.089} C_VEL
LIN {X 0,Y 146.822,Z 196.514,A -85,B 0,C 180,E1 -27211.282,E2 -27211.282} C_VEL
LIN {X 0,Y 149.347,Z 203.595,A -85,B 0,C 180,E1 -27213.466,E2 -27213.466} C_VEL
LIN {X 0,Y 151.847,Z 212.784,A -85,B 0,C 180,E1 -27215.856,E2 -27215.856} C_VEL
LIN {X 0,Y 154.867,Z 225.915,A -85,B 0,C 180,E1 -27219.443,E2 -27219.443} C_VEL
LIN {X 0,Y 157.351,Z 235.69,A -85,B 0,C 180,E1 -27222.529,E2 -27222.529} C_VEL
LIN {X 0,Y 159.876,Z 244.054,A -85,B 0,C 180,E1 -27225.496,E2 -27225.496} C_VEL
LIN {X 0,Y 163.202,Z 253.096,A -85,B 0,C 180,E1 -27229.089,E2 -27229.089} C_VEL
LIN {X 0,Y 167.366,Z 261.672,A -85,B 0,C 180,E1 -27232.922,E2 -27232.922} C_VEL
LIN {X 0,Y 172.875,Z 270.206,A -85,B 0,C 180,E1 -27237.179,E2 -27237.179} C_VEL
LIN {X 0,Y 179.179,Z 277.519,A -85,B 0,C 180,E1 -27241.202,E2 -27241.202} C_VEL
LIN {X 0,Y 186.189,Z 283.759,A -85,B 0,C 180,E1 -27244.944,E2 -27244.944} C_VEL
LIN {X 0,Y 195.642,Z 289.966,A -85,B 0,C 180,E1 -27249.063,E2 -27249.063} C_VEL
LIN {X 0,Y 205.992,Z 295.093,A -85,B 0,C 180,E1 -27252.8,E2 -27252.8} C_VEL
LIN {X 0,Y 217.139,Z 299.257,A -85,B 0,C 180,E1 -27256.161,E2 -27256.161} C_VEL
LIN {X 0,Y 228.898,Z 302.845,A -85,B 0,C 180,E1 -27259.384,E2 -27259.384} C_VEL
LIN {X 0,Y 236.533,Z 304.9,A -85,B 0,C 180,E1 -27261.456,E2 -27261.456} C_VEL
LIN {X 0,Y 242.871,Z 306.524,A -85,B 0,C 180,E1 -27263.353,E2 -27263.353} C_VEL
LIN {X 0,Y 248.066,Z 307.75,A -85,B 0,C 180,E1 -27265.124,E2 -27265.124} C_VEL
LIN {X 0,Y 253.213,Z 308.964,A -85,B 0,C 180,E1 -27267.669,E2 -27267.669} C_VEL
LIN {X 0,Y 254.323,Z 309.171,A -85,B 0,C 180,E1 -27268.416,E2 -27268.416} C_VEL
LIN {X 0,Y 255.854,Z 309.323,A -85,B 0,C 180,E1 -27270,E2 -27270} C_VEL
LIN {X 0,Y 254.323,Z 309.171,A -85,B 0,C 180,E1 -27271.584,E2 -27271.584} C_VEL
LIN {X 0,Y 251.524,Z 308.659,A -85,B 0,C 180,E1 -27273.204,E2 -27273.204} C_VEL
LIN {X 0,Y 248.063,Z 307.75,A -85,B 0,C 180,E1 -27274.876,E2 -27274.876} C_VEL
LIN {X 0,Y 240.879,Z 306.018,A -85,B 0,C 180,E1 -27277.261,E2 -27277.261} C_VEL
LIN {X 0,Y 234.813,Z 304.467,A -85,B 0,C 180,E1 -27279.004,E2 -27279.004} C_VEL
LIN {X 0,Y 222.912,Z 301.144,A -85,B 0,C 180,E1 -27282.217,E2 -27282.217} C_VEL
LIN {X 0,Y 208.714,Z 296.208,A -85,B 0,C 180,E1 -27286.33,E2 -27286.33} C_VEL
LIN {X 0,Y 198.142,Z 291.357,A -85,B 0,C 180,E1 -27289.962,E2 -27289.962} C_VEL
LIN {X 0,Y 187.692,Z 284.9,A -85,B 0,C 180,E1 -27294.323,E2 -27294.323} C_VEL
LIN {X 0,Y 180.963,Z 279.263,A -85,B 0,C 180,E1 -27297.777,E2 -27297.777} C_VEL
LIN {X 0,Y 174.845,Z 272.653,A -85,B 0,C 180,E1 -27301.503,E2 -27301.503} C_VEL
LIN {X 0,Y 169.238,Z 264.798,A -85,B 0,C 180,E1 -27305.548,E2 -27305.548} C_VEL
LIN {X 0,Y 165.127,Z 257.377,A -85,B 0,C 180,E1 -27309.039,E2 -27309.039} C_VEL
LIN {X 0,Y 161.764,Z 249.481,A -85,B 0,C 180,E1 -27312.391,E2 -27312.391} C_VEL
LIN {X 0,Y 158.487,Z 239.584,A -85,B 0,C 180,E1 -27316.109,E2 -27316.109} C_VEL
LIN {X 0,Y 155.933,Z 230.401,A -85,B 0,C 180,E1 -27319.196,E2 -27319.196} C_VEL
LIN {X 0,Y 153.455,Z 220.072,A -85,B 0,C 180,E1 -27322.227,E2 -27322.227} C_VEL
LIN {X 0,Y 150.824,Z 208.585,A -85,B 0,C 180,E1 -27325.195,E2 -27325.195} C_VEL
LIN {X 0,Y 147.735,Z 198.85,A -85,B 0,C 180,E1 -27327.925,E2 -27327.925} C_VEL
LIN {X 0,Y 144.355,Z 190.56,A -85,B 0,C 180,E1 -27330.977,E2 -27330.977} C_VEL
LIN {X 0,Y 140.79,Z 182.865,A -85,B 0,C 180,E1 -27334.623,E2 -27334.623} C_VEL
LIN {X 0,Y 137.734,Z 176.936,A -85,B 0,C 180,E1 -27338.29,E2 -27338.29} C_VEL
LIN {X 0,Y 135.82,Z 173.617,A -85,B 0,C 180,E1 -27340.966,E2 -27340.966} C_VEL
LIN {X 0,Y 134.093,Z 170.568,A -85,B 0,C 180,E1 -27343.835,E2 -27343.835} C_VEL
LIN {X 0,Y 131.974,Z 166.759,A -85,B 0,C 180,E1 -27348.435,E2 -27348.435} C_VEL
LIN {X 0,Y 130.127,Z 163.105,A -85,B 0,C 180,E1 -27355.937,E2 -27355.937} C_VEL
LIN {X 0,Y 129.973,Z 162.238,A -85,B 0,C 180,E1 -27358.452,E2 -27358.452} C_VEL
LIN {X 0,Y 129.991,Z 162.281,A -85,B 0,C 180,E1 -27361.551,E2 -27361.551} C_VEL
LIN {X 0,Y 130.204,Z 163.529,A -85,B 0,C 180,E1 -27364.452,E2 -27364.452} C_VEL
LIN {X 0,Y 132.325,Z 167.381,A -85,B 0,C 180,E1 -27372.077,E2 -27372.077} C_VEL
LIN {X 0,Y 134.701,Z 171.608,A -85,B 0,C 180,E1 -27376.854,E2 -27376.854} C_VEL
LIN {X 0,Y 137.002,Z 175.671,A -85,B 0,C 180,E1 -27380.359,E2 -27380.359} C_VEL
LIN {X 0,Y 139.68,Z 180.639,A -85,B 0,C 180,E1 -27383.737,E2 -27383.737} C_VEL
LIN {X 0,Y 141.772,Z 186.172,A -85,B 0,C 180,E1 -27386.202,E2 -27386.202} C_VEL
LIN {X 0,Y 144.445,Z 194.617,A -85,B 0,C 180,E1 -27389.116,E2 -27389.116} C_VEL
LIN {X 0,Y 142.368,Z 215.271,A -85,B 0,C 180,E1 -27389.926,E2 -27389.926} C_VEL
LIN {X 0,Y 139.745,Z 228.957,A -85,B 0,C 180,E1 -27390.737,E2 -27390.737} C_VEL
LIN {X 0,Y 136.392,Z 240.462,A -85,B 0,C 180,E1 -27391.766,E2 -27391.766} C_VEL
LIN {X 0,Y 132.885,Z 249.972,A -85,B 0,C 180,E1 -27392.903,E2 -27392.903} C_VEL
LIN {X 0,Y 128.776,Z 259.242,A -85,B 0,C 180,E1 -27394.366,E2 -27394.366} C_VEL
LIN {X 0,Y 124.105,Z 268.181,A -85,B 0,C 180,E1 -27396.199,E2 -27396.199} C_VEL
LIN {X 0,Y 118.938,Z 276.702,A -85,B 0,C 180,E1 -27398.47,E2 -27398.47} C_VEL
LIN {X 0,Y 114.018,Z 283.916,A -85,B 0,C 180,E1 -27400.968,E2 -27400.968} C_VEL
LIN {X 0,Y 109.353,Z 290.114,A -85,B 0,C 180,E1 -27403.695,E2 -27403.695} C_VEL
LIN {X 0,Y 103.941,Z 296.648,A -85,B 0,C 180,E1 -27407.456,E2 -27407.456} C_VEL
LIN {X 0,Y 100.046,Z 301.152,A -85,B 0,C 180,E1 -27410.786,E2 -27410.786} C_VEL
LIN {X 0,Y 94.751,Z 306.643,A -85,B 0,C 180,E1 -27416.2,E2 -27416.2} C_VEL
LIN {X 0,Y 90.368,Z 310.971,A -85,B 0,C 180,E1 -27422.185,E2 -27422.185} C_VEL
LIN {X 0,Y 87.975,Z 313.34,A -85,B 0,C 180,E1 -27426.457,E2 -27426.457} C_VEL
LIN {X 0,Y 86.22,Z 315.146,A -85,B 0,C 180,E1 -27430.971,E2 -27430.971} C_VEL
LIN {X 0,Y 84.145,Z 317.61,A -85,B 0,C 180,E1 -27440.384,E2 -27440.384} C_VEL
LIN {X 0,Y 83.796,Z 318.207,A -85,B 0,C 180,E1 -27445.189,E2 -27445.189} C_VEL
LIN {X 0,Y 83.883,Z 318.37,A -85,B 0,C 180,E1 -27450,E2 -27450} C_VEL
LIN {X 0,Y 83.79,Z 318.207,A -85,B 0,C 180,E1 -27454.811,E2 -27454.811} C_VEL
LIN {X 0,Y 84.131,Z 317.609,A -85,B 0,C 180,E1 -27459.618,E2 -27459.618} C_VEL
LIN {X 0,Y 86.22,Z 315.146,A -85,B 0,C 180,E1 -27469.029,E2 -27469.029} C_VEL
LIN {X 0,Y 89.113,Z 312.188,A -85,B 0,C 180,E1 -27475.706,E2 -27475.706} C_VEL
LIN {X 0,Y 93.18,Z 308.198,A -85,B 0,C 180,E1 -27481.868,E2 -27481.868} C_VEL
LIN {X 0,Y 98.256,Z 303.07,A -85,B 0,C 180,E1 -27487.444,E2 -27487.444} C_VEL
LIN {X 0,Y 102.55,Z 298.325,A -85,B 0,C 180,E1 -27491.338,E2 -27491.338} C_VEL
LIN {X 0,Y 108.243,Z 291.489,A -85,B 0,C 180,E1 -27495.578,E2 -27495.578} C_VEL
LIN {X 0,Y 112.851,Z 285.543,A -85,B 0,C 180,E1 -27498.359,E2 -27498.359} C_VEL
LIN {X 0,Y 117.717,Z 278.621,A -85,B 0,C 180,E1 -27500.908,E2 -27500.908} C_VEL
LIN {X 0,Y 122.794,Z 270.448,A -85,B 0,C 180,E1 -27503.252,E2 -27503.252} C_VEL
LIN {X 0,Y 127.416,Z 261.942,A -85,B 0,C 180,E1 -27505.132,E2 -27505.132} C_VEL
LIN {X 0,Y 131.486,Z 253.233,A -85,B 0,C 180,E1 -27506.633,E2 -27506.633} C_VEL
LIN {X 0,Y 135.347,Z 243.482,A -85,B 0,C 180,E1 -27507.891,E2 -27507.891} C_VEL
LIN {X 0,Y 138.512,Z 233.404,A -85,B 0,C 180,E1 -27508.895,E2 -27508.895} C_VEL
LIN {X 0,Y 140.956,Z 223.123,A -85,B 0,C 180,E1 -27509.656,E2 -27509.656} C_VEL
LIN {X 0,Y 142.604,Z 213.224,A -85,B 0,C 180,E1 -27510.168,E2 -27510.168} C_VEL
LIN {X 0,Y 144.389,Z 194.499,A -85,B 0,C 180,E1 -27510.935,E2 -27510.935} C_VEL
LIN {X 0,Y 141.257,Z 184.716,A -85,B 0,C 180,E1 -27514.389,E2 -27514.389} C_VEL
LIN {X 0,Y 139.385,Z 180.066,A -85,B 0,C 180,E1 -27516.609,E2 -27516.609} C_VEL
LIN {X 0,Y 136.328,Z 174.337,A -85,B 0,C 180,E1 -27520.616,E2 -27520.616} C_VEL
LIN {X 0,Y 133.991,Z 170.364,A -85,B 0,C 180,E1 -27524.405,E2 -27524.405} C_VEL
LIN {X 0,Y 132.069,Z 166.847,A -85,B 0,C 180,E1 -27528.587,E2 -27528.587} C_VEL
LIN {X 0,Y 130.033,Z 162.464,A -85,B 0,C 180,E1 -27537.675,E2 -27537.675} C_VEL
LIN {X 0,Y 129.956,Z 162.083,A -85,B 0,C 180,E1 -27539.998,E2 -27539.998} C_VEL
LIN {X 0,Y 130.089,Z 162.739,A -85,B 0,C 180,E1 -27543.483,E2 -27543.483} C_VEL
LIN {X 0,Y 131.829,Z 166.632,A -85,B 0,C 180,E1 -27551.212,E2 -27551.212} C_VEL
LIN {X 0,Y 132.38,Z 167.533,A -85,B 0,C 180,E1 -27552.601,E2 -27552.601} C_VEL
LIN {X 0,Y 134.822,Z 171.839,A -85,B 0,C 180,E1 -27557.44,E2 -27557.44} C_VEL
LIN {X 0,Y 136.438,Z 174.52,A -85,B 0,C 180,E1 -27559.918,E2 -27559.918} C_VEL
LIN {X 0,Y 137.212,Z 177.013,A -85,B 0,C 180,E1 -27561.161,E2 -27561.161} C_VEL
LIN {X 0,Y 137.945,Z 182.578,A -85,B 0,C 180,E1 -27562.695,E2 -27562.695} C_VEL
LIN {X 0,Y 138.7,Z 188.337,A -85,B 0,C 180,E1 -27564.166,E2 -27564.166} C_VEL
LIN {X 0,Y 139.584,Z 191.126,A -85,B 0,C 180,E1 -27565.302,E2 -27565.302} C_VEL
LIN {X 0,Y 143.021,Z 199.426,A -85,B 0,C 180,E1 -27568.955,E2 -27568.955} C_VEL
LIN {X 0,Y 145.668,Z 207.436,A -85,B 0,C 180,E1 -27571.645,E2 -27571.645} C_VEL
LIN {X 0,Y 147.659,Z 215.948,A -85,B 0,C 180,E1 -27574.002,E2 -27574.002} C_VEL
LIN {X 0,Y 149.638,Z 226.495,A -85,B 0,C 180,E1 -27577.02,E2 -27577.02} C_VEL
LIN {X 0,Y 151.472,Z 235.829,A -85,B 0,C 180,E1 -27580.019,E2 -27580.019} C_VEL
LIN {X 0,Y 153.633,Z 244.85,A -85,B 0,C 180,E1 -27583.326,E2 -27583.326} C_VEL
LIN {X 0,Y 156.375,Z 253.704,A -85,B 0,C 180,E1 -27587.006,E2 -27587.006} C_VEL
LIN {X 0,Y 159.467,Z 261.625,A -85,B 0,C 180,E1 -27590.633,E2 -27590.633} C_VEL
LIN {X 0,Y 164.4,Z 270.472,A -85,B 0,C 180,E1 -27595.252,E2 -27595.252} C_VEL
LIN {X 0,Y 170.009,Z 277.81,A -85,B 0,C 180,E1 -27599.495,E2 -27599.495} C_VEL
LIN {X 0,Y 176.234,Z 283.929,A -85,B 0,C 180,E1 -27603.365,E2 -27603.365} C_VEL
LIN {X 0,Y 184.629,Z 290.04,A -85,B 0,C 180,E1 -27607.626,E2 -27607.626} C_VEL
LIN {X 0,Y 195.686,Z 295.827,A -85,B 0,C 180,E1 -27612.123,E2 -27612.123} C_VEL
LIN {X 0,Y 208.777,Z 300.67,A -85,B 0,C 180,E1 -27616.371,E2 -27616.371} C_VEL
LIN {X 0,Y 221.305,Z 304.157,A -85,B 0,C 180,E1 -27619.883,E2 -27619.883} C_VEL
LIN {X 0,Y 227.384,Z 305.568,A -85,B 0,C 180,E1 -27621.509,E2 -27621.509} C_VEL
LIN {X 0,Y 233.542,Z 306.914,A -85,B 0,C 180,E1 -27623.242,E2 -27623.242} C_VEL
LIN {X 0,Y 239.785,Z 308.149,A -85,B 0,C 180,E1 -27625.211,E2 -27625.211} C_VEL
LIN {X 0,Y 243.449,Z 308.878,A -85,B 0,C 180,E1 -27626.69,E2 -27626.69} C_VEL
LIN {X 0,Y 246.775,Z 309.373,A -85,B 0,C 180,E1 -27628.368,E2 -27628.368} C_VEL
LIN {X 0,Y 248.597,Z 309.514,A -85,B 0,C 180,E1 -27630,E2 -27630} C_VEL
LIN {X 0,Y 246.768,Z 309.373,A -85,B 0,C 180,E1 -27631.632,E2 -27631.632} C_VEL
LIN {X 0,Y 243.441,Z 308.878,A -85,B 0,C 180,E1 -27633.31,E2 -27633.31} C_VEL
LIN {X 0,Y 238.961,Z 307.993,A -85,B 0,C 180,E1 -27635.062,E2 -27635.062} C_VEL
LIN {X 0,Y 232.925,Z 306.794,A -85,B 0,C 180,E1 -27636.932,E2 -27636.932} C_VEL
LIN {X 0,Y 225.541,Z 305.198,A -85,B 0,C 180,E1 -27638.963,E2 -27638.963} C_VEL
LIN {X 0,Y 215.345,Z 302.623,A -85,B 0,C 180,E1 -27641.746,E2 -27641.746} C_VEL
LIN {X 0,Y 200.186,Z 297.745,A -85,B 0,C 180,E1 -27646.311,E2 -27646.311} C_VEL
LIN {X 0,Y 188.023,Z 292.081,A -85,B 0,C 180,E1 -27650.863,E2 -27650.863} C_VEL
LIN {X 0,Y 178.724,Z 285.967,A -85,B 0,C 180,E1 -27655.256,E2 -27655.256} C_VEL
LIN {X 0,Y 171.621,Z 279.541,A -85,B 0,C 180,E1 -27659.433,E2 -27659.433} C_VEL
LIN {X 0,Y 165.627,Z 272.211,A -85,B 0,C 180,E1 -27663.76,E2 -27663.76} C_VEL
LIN {X 0,Y 161.176,Z 265.059,A -85,B 0,C 180,E1 -27667.623,E2 -27667.623} C_VEL
LIN {X 0,Y 158.074,Z 258.367,A -85,B 0,C 180,E1 -27670.905,E2 -27670.905} C_VEL
LIN {X 0,Y 155.281,Z 250.4,A -85,B 0,C 180,E1 -27674.423,E2 -27674.423} C_VEL
LIN {X 0,Y 152.709,Z 240.9,A -85,B 0,C 180,E1 -27678.14,E2 -27678.14} C_VEL
LIN {X 0,Y 150.597,Z 231.457,A -85,B 0,C 180,E1 -27681.431,E2 -27681.431} C_VEL
LIN {X 0,Y 148.389,Z 220.175,A -85,B 0,C 180,E1 -27684.85,E2 -27684.85} C_VEL
LIN {X 0,Y 146.391,Z 210.015,A -85,B 0,C 180,E1 -27687.618,E2 -27687.618} C_VEL
LIN {X 0,Y 143.908,Z 201.866,A -85,B 0,C 180,E1 -27690.165,E2 -27690.165} C_VEL
LIN {X 0,Y 140.516,Z 193.311,A -85,B 0,C 180,E1 -27693.65,E2 -27693.65} C_VEL
LIN {X 0,Y 137.406,Z 186.334,A -85,B 0,C 180,E1 -27697.345,E2 -27697.345} C_VEL
LIN {X 0,Y 134.44,Z 180.489,A -85,B 0,C 180,E1 -27701.585,E2 -27701.585} C_VEL
LIN {X 0,Y 132.424,Z 176.836,A -85,B 0,C 180,E1 -27705.204,E2 -27705.204} C_VEL
LIN {X 0,Y 130.83,Z 173.631,A -85,B 0,C 180,E1 -27709.069,E2 -27709.069} C_VEL
LIN {X 0,Y 129.138,Z 169.475,A -85,B 0,C 180,E1 -27717.662,E2 -27717.662} C_VEL
LIN {X 0,Y 129.098,Z 169.216,A -85,B 0,C 180,E1 -27720.781,E2 -27720.781} C_VEL
LIN {X 0,Y 129.224,Z 170.228,A -85,B 0,C 180,E1 -27723.509,E2 -27723.509} C_VEL
LIN {X 0,Y 131.053,Z 174.075,A -85,B 0,C 180,E1 -27731.177,E2 -27731.177} C_VEL
LIN {X 0,Y 133.285,Z 178.389,A -85,B 0,C 180,E1 -27736.073,E2 -27736.073} C_VEL
LIN {X 0,Y 135.216,Z 182.036,A -85,B 0,C 180,E1 -27739.254,E2 -27739.254} C_VEL
LIN {X 0,Y 137.691,Z 187.014,A -85,B 0,C 180,E1 -27742.653,E2 -27742.653} C_VEL
LIN {X 0,Y 139.786,Z 193.673,A -85,B 0,C 180,E1 -27745.399,E2 -27745.399} C_VEL
LIN {X 0,Y 140.84,Z 197.335,A -85,B 0,C 180,E1 -27746.688,E2 -27746.688} C_VEL
LIN {X 0,Y 138.701,Z 216.937,A -85,B 0,C 180,E1 -27747.469,E2 -27747.469} C_VEL
LIN {X 0,Y 135.709,Z 230.639,A -85,B 0,C 180,E1 -27748.311,E2 -27748.311} C_VEL
LIN {X 0,Y 132.42,Z 241.278,A -85,B 0,C 180,E1 -27749.262,E2 -27749.262} C_VEL
LIN {X 0,Y 128.447,Z 251.412,A -85,B 0,C 180,E1 -27750.485,E2 -27750.485} C_VEL
LIN {X 0,Y 124.192,Z 260.401,A -85,B 0,C 180,E1 -27751.914,E2 -27751.914} C_VEL
LIN {X 0,Y 119.367,Z 269.124,A -85,B 0,C 180,E1 -27753.732,E2 -27753.732} C_VEL
LIN {X 0,Y 114.653,Z 276.511,A -85,B 0,C 180,E1 -27755.689,E2 -27755.689} C_VEL
LIN {X 0,Y 109.49,Z 283.725,A -85,B 0,C 180,E1 -27758.159,E2 -27758.159} C_VEL
LIN {X 0,Y 104.571,Z 289.923,A -85,B 0,C 180,E1 -27760.88,E2 -27760.88} C_VEL
LIN {X 0,Y 98.799,Z 296.457,A -85,B 0,C 180,E1 -27764.656,E2 -27764.656} C_VEL
LIN {X 0,Y 94.62,Z 300.96,A -85,B 0,C 180,E1 -27768.05,E2 -27768.05} C_VEL
LIN {X 0,Y 88.923,Z 306.452,A -85,B 0,C 180,E1 -27773.647,E2 -27773.647} C_VEL
LIN {X 0,Y 84.127,Z 310.779,A -85,B 0,C 180,E1 -27779.918,E2 -27779.918} C_VEL
LIN {X 0,Y 81.483,Z 313.148,A -85,B 0,C 180,E1 -27784.453,E2 -27784.453} C_VEL
LIN {X 0,Y 79.503,Z 314.955,A -85,B 0,C 180,E1 -27789.293,E2 -27789.293} C_VEL
LIN {X 0,Y 77.13,Z 317.418,A -85,B 0,C 180,E1 -27799.5,E2 -27799.5} C_VEL
LIN {X 0,Y 76.733,Z 318.017,A -85,B 0,C 180,E1 -27804.745,E2 -27804.745} C_VEL
LIN {X 0,Y 76.781,Z 318.179,A -85,B 0,C 180,E1 -27810,E2 -27810} C_VEL
LIN {X 0,Y 76.71,Z 318.016,A -85,B 0,C 180,E1 -27815.257,E2 -27815.257} C_VEL
LIN {X 0,Y 77.119,Z 317.418,A -85,B 0,C 180,E1 -27820.502,E2 -27820.502} C_VEL
LIN {X 0,Y 79.503,Z 314.955,A -85,B 0,C 180,E1 -27830.707,E2 -27830.707} C_VEL
LIN {X 0,Y 82.751,Z 311.997,A -85,B 0,C 180,E1 -27837.847,E2 -27837.847} C_VEL
LIN {X 0,Y 87.196,Z 308.006,A -85,B 0,C 180,E1 -27844.347,E2 -27844.347} C_VEL
LIN {X 0,Y 92.694,Z 302.878,A -85,B 0,C 180,E1 -27850.125,E2 -27850.125} C_VEL
LIN {X 0,Y 97.775,Z 297.616,A -85,B 0,C 180,E1 -27854.491,E2 -27854.491} C_VEL
LIN {X 0,Y 103.374,Z 291.298,A -85,B 0,C 180,E1 -27858.404,E2 -27858.404} C_VEL
LIN {X 0,Y 108.254,Z 285.352,A -85,B 0,C 180,E1 -27861.174,E2 -27861.174} C_VEL
LIN {X 0,Y 113.373,Z 278.431,A -85,B 0,C 180,E1 -27863.694,E2 -27863.694} C_VEL
LIN {X 0,Y 118.675,Z 270.257,A -85,B 0,C 180,E1 -27866.005,E2 -27866.005} C_VEL
LIN {X 0,Y 123.499,Z 261.752,A -85,B 0,C 180,E1 -27867.833,E2 -27867.833} C_VEL
LIN {X 0,Y 127.725,Z 253.042,A -85,B 0,C 180,E1 -27869.289,E2 -27869.289} C_VEL
LIN {X 0,Y 131.717,Z 243.292,A -85,B 0,C 180,E1 -27870.503,E2 -27870.503} C_VEL
LIN {X 0,Y 134.627,Z 234.502,A -85,B 0,C 180,E1 -27871.362,E2 -27871.362} C_VEL
LIN {X 0,Y 137.263,Z 224.053,A -85,B 0,C 180,E1 -27872.149,E2 -27872.149} C_VEL
LIN {X 0,Y 139.089,Z 213.894,A -85,B 0,C 180,E1 -27872.672,E2 -27872.672} C_VEL
LIN {X 0,Y 140.847,Z 197.276,A -85,B 0,C 180,E1 -27873.313,E2 -27873.313} C_VEL
LIN {X 0,Y 138.273,Z 188.664,A -85,B 0,C 180,E1 -27876.571,E2 -27876.571} C_VEL
LIN {X 0,Y 136.85,Z 185.252,A -85,B 0,C 180,E1 -27878.442,E2 -27878.442} C_VEL
LIN {X 0,Y 134.241,Z 180.137,A -85,B 0,C 180,E1 -27882.282,E2 -27882.282} C_VEL
LIN {X 0,Y 132.331,Z 176.635,A -85,B 0,C 180,E1 -27885.779,E2 -27885.779} C_VEL
LIN {X 0,Y 130.739,Z 173.506,A -85,B 0,C 180,E1 -27889.696,E2 -27889.696} C_VEL
LIN {X 0,Y 129.12,Z 169.375,A -85,B 0,C 180,E1 -27898.439,E2 -27898.439} C_VEL
LIN {X 0,Y 129.091,Z 169.129,A -85,B 0,C 180,E1 -27899.998,E2 -27899.998} C_VEL
LIN {X 0,Y 129.175,Z 169.812,A -85,B 0,C 180,E1 -27903.117,E2 -27903.117} C_VEL
LIN {X 0,Y 130.708,Z 173.508,A -85,B 0,C 180,E1 -27910.609,E2 -27910.609} C_VEL
LIN {X 0,Y 131.724,Z 175.643,A -85,B 0,C 180,E1 -27913.301,E2 -27913.301} C_VEL
LIN {X 0,Y 133.243,Z 178.292,A -85,B 0,C 180,E1 -27916.369,E2 -27916.369} C_VEL
LIN {X 0,Y 135.156,Z 181.919,A -85,B 0,C 180,E1 -27919.541,E2 -27919.541} C_VEL
LIN {X 0,Y 137.728,Z 187.044,A -85,B 0,C 180,E1 -27923.07,E2 -27923.07} C_VEL
LIN {X 0,Y 139.584,Z 191.126,A -85,B 0,C 180,E1 -27925.302,E2 -27925.302} C_VEL
LIN {X 0,Y 140.59,Z 193.693,A -85,B 0,C 180,E1 -27926.444,E2 -27926.444} C_VEL
LIN {X 0,Y 141.693,Z 198.416,A -85,B 0,C 180,E1 -27927.821,E2 -27927.821} C_VEL
LIN {X 0,Y 142.373,Z 203.689,A -85,B 0,C 180,E1 -27928.918,E2 -27928.918} C_VEL
LIN {X 0,Y 143.2,Z 214.799,A -85,B 0,C 180,E1 -27930.993,E2 -27930.993} C_VEL
LIN {X 0,Y 143.454,Z 218.285,A -85,B 0,C 180,E1 -27931.837,E2 -27931.837} C_VEL
LIN {X 0,Y 144.808,Z 227.868,A -85,B 0,C 180,E1 -27934.683,E2 -27934.683} C_VEL
LIN {X 0,Y 146.267,Z 237.803,A -85,B 0,C 180,E1 -27938.022,E2 -27938.022} C_VEL
LIN {X 0,Y 147.655,Z 245.302,A -85,B 0,C 180,E1 -27940.877,E2 -27940.877} C_VEL
LIN {X 0,Y 149.793,Z 254.274,A -85,B 0,C 180,E1 -27944.728,E2 -27944.728} C_VEL
LIN {X 0,Y 152.602,Z 262.973,A -85,B 0,C 180,E1 -27948.924,E2 -27948.924} C_VEL
LIN {X 0,Y 156.321,Z 270.779,A -85,B 0,C 180,E1 -27953.192,E2 -27953.192} C_VEL
LIN {X 0,Y 161.153,Z 278.088,A -85,B 0,C 180,E1 -27957.626,E2 -27957.626} C_VEL
LIN {X 0,Y 167.155,Z 284.596,A -85,B 0,C 180,E1 -27961.996,E2 -27961.996} C_VEL
LIN {X 0,Y 174.302,Z 290.335,A -85,B 0,C 180,E1 -27966.221,E2 -27966.221} C_VEL
LIN {X 0,Y 181.327,Z 294.529,A -85,B 0,C 180,E1 -27969.584,E2 -27969.584} C_VEL
LIN {X 0,Y 190.715,Z 298.778,A -85,B 0,C 180,E1 -27973.356,E2 -27973.356} C_VEL
LIN {X 0,Y 205.706,Z 303.467,A -85,B 0,C 180,E1 -27978.171,E2 -27978.171} C_VEL
LIN {X 0,Y 214.26,Z 305.505,A -85,B 0,C 180,E1 -27980.561,E2 -27980.561} C_VEL
LIN {X 0,Y 222.378,Z 307.08,A -85,B 0,C 180,E1 -27982.738,E2 -27982.738} C_VEL
LIN {X 0,Y 229.312,Z 308.25,A -85,B 0,C 180,E1 -27984.725,E2 -27984.725} C_VEL
LIN {X 0,Y 232.567,Z 308.773,A -85,B 0,C 180,E1 -27985.725,E2 -27985.725} C_VEL
LIN {X 0,Y 234.895,Z 309.109,A -85,B 0,C 180,E1 -27986.569,E2 -27986.569} C_VEL
LIN {X 0,Y 239.041,Z 309.604,A -85,B 0,C 180,E1 -27988.396,E2 -27988.396} C_VEL
LIN {X 0,Y 241.248,Z 309.707,A -85,B 0,C 180,E1 -27990,E2 -27990} C_VEL
LIN {X 0,Y 238.868,Z 309.584,A -85,B 0,C 180,E1 -27991.686,E2 -27991.686} C_VEL
LIN {X 0,Y 234.892,Z 309.109,A -85,B 0,C 180,E1 -27993.431,E2 -27993.431} C_VEL
LIN {X 0,Y 232.566,Z 308.774,A -85,B 0,C 180,E1 -27994.274,E2 -27994.274} C_VEL
LIN {X 0,Y 226.205,Z 307.781,A -85,B 0,C 180,E1 -27996.178,E2 -27996.178} C_VEL
LIN {X 0,Y 219.947,Z 306.634,A -85,B 0,C 180,E1 -27997.893,E2 -27997.893} C_VEL
LIN {X 0,Y 207.777,Z 304.003,A -85,B 0,C 180,E1 -28001.218,E2 -28001.218} C_VEL
LIN {X 0,Y 196.197,Z 300.718,A -85,B 0,C 180,E1 -28004.727,E2 -28004.727} C_VEL
LIN {X 0,Y 185.442,Z 296.509,A -85,B 0,C 180,E1 -28008.658,E2 -28008.658} C_VEL
LIN {X 0,Y 175.669,Z 291.254,A -85,B 0,C 180,E1 -28013.053,E2 -28013.053} C_VEL
LIN {X 0,Y 168.118,Z 285.47,A -85,B 0,C 180,E1 -28017.377,E2 -28017.377} C_VEL
LIN {X 0,Y 162.639,Z 279.813,A -85,B 0,C 180,E1 -28021.235,E2 -28021.235} C_VEL
LIN {X 0,Y 157.753,Z 273.186,A -85,B 0,C 180,E1 -28025.391,E2 -28025.391} C_VEL
LIN {X 0,Y 154.14,Z 266.555,A -85,B 0,C 180,E1 -28029.187,E2 -28029.187} C_VEL
LIN {X 0,Y 150.726,Z 257.621,A -85,B 0,C 180,E1 -28033.724,E2 -28033.724} C_VEL
LIN {X 0,Y 148.443,Z 248.965,A -85,B 0,C 180,E1 -28037.6,E2 -28037.6} C_VEL
LIN {X 0,Y 146.541,Z 239.257,A -85,B 0,C 180,E1 -28041.432,E2 -28041.432} C_VEL
LIN {X 0,Y 145.196,Z 230.398,A -85,B 0,C 180,E1 -28044.492,E2 -28044.492} C_VEL
LIN {X 0,Y 143.807,Z 220.663,A -85,B 0,C 180,E1 -28047.483,E2 -28047.483} C_VEL
LIN {X 0,Y 142.204,Z 211.655,A -85,B 0,C 180,E1 -28050.18,E2 -28050.18} C_VEL
LIN {X 0,Y 140.388,Z 205.202,A -85,B 0,C 180,E1 -28052.417,E2 -28052.417} C_VEL
LIN {X 0,Y 137.248,Z 196.893,A -85,B 0,C 180,E1 -28056.12,E2 -28056.12} C_VEL
LIN {X 0,Y 134.579,Z 190.699,A -85,B 0,C 180,E1 -28059.784,E2 -28059.784} C_VEL
LIN {X 0,Y 132.479,Z 186.36,A -85,B 0,C 180,E1 -28063.236,E2 -28063.236} C_VEL
LIN {X 0,Y 130.918,Z 183.239,A -85,B 0,C 180,E1 -28066.418,E2 -28066.418} C_VEL
LIN {X 0,Y 129.614,Z 180.394,A -85,B 0,C 180,E1 -28069.971,E2 -28069.971} C_VEL
LIN {X 0,Y 128.236,Z 176.388,A -85,B 0,C 180,E1 -28078.431,E2 -28078.431} C_VEL
LIN {X 0,Y 128.239,Z 176.355,A -85,B 0,C 180,E1 -28081.179,E2 -28081.179} C_VEL
LIN {X 0,Y 129.868,Z 180.928,A -85,B 0,C 180,E1 -28090.436,E2 -28090.436} C_VEL
LIN {X 0,Y 131.843,Z 185.016,A -85,B 0,C 180,E1 -28095.163,E2 -28095.163} C_VEL
LIN {X 0,Y 134.057,Z 189.519,A -85,B 0,C 180,E1 -28099.029,E2 -28099.029} C_VEL
LIN {X 0,Y 135.677,Z 193.425,A -85,B 0,C 180,E1 -28101.46,E2 -28101.46} C_VEL
LIN {X 0,Y 137.5,Z 200.058,A -85,B 0,C 180,E1 -28104.137,E2 -28104.137} C_VEL
LIN {X 0,Y 135.403,Z 217.816,A -85,B 0,C 180,E1 -28104.853,E2 -28104.853} C_VEL
LIN {X 0,Y 132.497,Z 230.449,A -85,B 0,C 180,E1 -28105.615,E2 -28105.615} C_VEL
LIN {X 0,Y 129.101,Z 241.087,A -85,B 0,C 180,E1 -28106.515,E2 -28106.515} C_VEL
LIN {X 0,Y 125.003,Z 251.222,A -85,B 0,C 180,E1 -28107.686,E2 -28107.686} C_VEL
LIN {X 0,Y 120.593,Z 260.211,A -85,B 0,C 180,E1 -28109.052,E2 -28109.052} C_VEL
LIN {X 0,Y 115.572,Z 268.933,A -85,B 0,C 180,E1 -28110.802,E2 -28110.802} C_VEL
LIN {X 0,Y 110.656,Z 276.321,A -85,B 0,C 180,E1 -28112.698,E2 -28112.698} C_VEL
LIN {X 0,Y 105.236,Z 283.534,A -85,B 0,C 180,E1 -28115.106,E2 -28115.106} C_VEL
LIN {X 0,Y 100.052,Z 289.732,A -85,B 0,C 180,E1 -28117.792,E2 -28117.792} C_VEL
LIN {X 0,Y 93.924,Z 296.265,A -85,B 0,C 180,E1 -28121.56,E2 -28121.56} C_VEL
LIN {X 0,Y 88.209,Z 301.868,A -85,B 0,C 180,E1 -28126.035,E2 -28126.035} C_VEL
LIN {X 0,Y 83.3,Z 306.261,A -85,B 0,C 180,E1 -28130.745,E2 -28130.745} C_VEL
LIN {X 0,Y 78.043,Z 310.588,A -85,B 0,C 180,E1 -28137.295,E2 -28137.295} C_VEL
LIN {X 0,Y 75.113,Z 312.957,A -85,B 0,C 180,E1 -28142.107,E2 -28142.107} C_VEL
LIN {X 0,Y 72.875,Z 314.763,A -85,B 0,C 180,E1 -28147.31,E2 -28147.31} C_VEL
LIN {X 0,Y 70.148,Z 317.228,A -85,B 0,C 180,E1 -28158.441,E2 -28158.441} C_VEL
LIN {X 0,Y 69.645,Z 317.826,A -85,B 0,C 180,E1 -28164.208,E2 -28164.208} C_VEL
LIN {X 0,Y 69.677,Z 317.988,A -85,B 0,C 180,E1 -28170,E2 -28170} C_VEL
LIN {X 0,Y 69.623,Z 317.825,A -85,B 0,C 180,E1 -28175.794,E2 -28175.794} C_VEL
LIN {X 0,Y 70.118,Z 317.227,A -85,B 0,C 180,E1 -28181.564,E2 -28181.564} C_VEL
LIN {X 0,Y 72.875,Z 314.763,A -85,B 0,C 180,E1 -28192.691,E2 -28192.691} C_VEL
LIN {X 0,Y 76.526,Z 311.806,A -85,B 0,C 180,E1 -28200.338,E2 -28200.338} C_VEL
LIN {X 0,Y 81.404,Z 307.815,A -85,B 0,C 180,E1 -28207.181,E2 -28207.181} C_VEL
LIN {X 0,Y 87.344,Z 302.686,A -85,B 0,C 180,E1 -28213.152,E2 -28213.152} C_VEL
LIN {X 0,Y 92.819,Z 297.424,A -85,B 0,C 180,E1 -28217.58,E2 -28217.58} C_VEL
LIN {X 0,Y 98.796,Z 291.107,A -85,B 0,C 180,E1 -28221.49,E2 -28221.49} C_VEL
LIN {X 0,Y 103.939,Z 285.161,A -85,B 0,C 180,E1 -28224.232,E2 -28224.232} C_VEL
LIN {X 0,Y 109.303,Z 278.239,A -85,B 0,C 180,E1 -28226.707,E2 -28226.707} C_VEL
LIN {X 0,Y 114.856,Z 270.067,A -85,B 0,C 180,E1 -28228.943,E2 -28228.943} C_VEL
LIN {X 0,Y 119.874,Z 261.562,A -85,B 0,C 180,E1 -28230.703,E2 -28230.703} C_VEL
LIN {X 0,Y 124.257,Z 252.852,A -85,B 0,C 180,E1 -28232.098,E2 -28232.098} C_VEL
LIN {X 0,Y 128.377,Z 243.102,A -85,B 0,C 180,E1 -28233.256,E2 -28233.256} C_VEL
LIN {X 0,Y 131.375,Z 234.311,A -85,B 0,C 180,E1 -28234.078,E2 -28234.078} C_VEL
LIN {X 0,Y 134.082,Z 223.947,A -85,B 0,C 180,E1 -28234.822,E2 -28234.822} C_VEL
LIN {X 0,Y 135.95,Z 213.935,A -85,B 0,C 180,E1 -28235.316,E2 -28235.316} C_VEL
LIN {X 0,Y 137.502,Z 200.044,A -85,B 0,C 180,E1 -28235.863,E2 -28235.863} C_VEL
LIN {X 0,Y 135.62,Z 193.21,A -85,B 0,C 180,E1 -28238.631,E2 -28238.631} C_VEL
LIN {X 0,Y 133.595,Z 188.606,A -85,B 0,C 180,E1 -28241.698,E2 -28241.698} C_VEL
LIN {X 0,Y 131.36,Z 183.88,A -85,B 0,C 180,E1 -28245.87,E2 -28245.87} C_VEL
LIN {X 0,Y 129.656,Z 180.394,A -85,B 0,C 180,E1 -28250.241,E2 -28250.241} C_VEL
LIN {X 0,Y 128.252,Z 176.444,A -85,B 0,C 180,E1 -28258.428,E2 -28258.428} C_VEL
LIN {X 0,Y 128.224,Z 176.187,A -85,B 0,C 180,E1 -28259.998,E2 -28259.998} C_VEL
LIN {X 0,Y 128.262,Z 176.762,A -85,B 0,C 180,E1 -28262.55,E2 -28262.55} C_VEL
LIN {X 0,Y 129.879,Z 180.94,A -85,B 0,C 180,E1 -28270.844,E2 -28270.844} C_VEL
LIN {X 0,Y 131.849,Z 185.046,A -85,B 0,C 180,E1 -28275.554,E2 -28275.554} C_VEL
LIN {X 0,Y 134.136,Z 189.69,A -85,B 0,C 180,E1 -28279.531,E2 -28279.531} C_VEL
LIN {X 0,Y 136.752,Z 195.684,A -85,B 0,C 180,E1 -28283.244,E2 -28283.244} C_VEL
LIN {X 0,Y 139.864,Z 203.714,A -85,B 0,C 180,E1 -28286.986,E2 -28286.986} C_VEL
LIN {X 0,Y 142.111,Z 211.327,A -85,B 0,C 180,E1 -28289.74,E2 -28289.74} C_VEL
LIN {X 0,Y 143.454,Z 218.285,A -85,B 0,C 180,E1 -28291.837,E2 -28291.837} C_VEL
LIN {X 0,Y 143.789,Z 223.415,A -85,B 0,C 180,E1 -28293.022,E2 -28293.022} C_VEL
LIN {X 0,Y 142.965,Z 232.402,A -85,B 0,C 180,E1 -28294.7,E2 -28294.7} C_VEL
LIN {X 0,Y 141.96,Z 240.977,A -85,B 0,C 180,E1 -28296.605,E2 -28296.605} C_VEL
LIN {X 0,Y 141.983,Z 245.458,A -85,B 0,C 180,E1 -28298.127,E2 -28298.127} C_VEL
LIN {X 0,Y 143.602,Z 255.297,A -85,B 0,C 180,E1 -28302.484,E2 -28302.484} C_VEL
LIN {X 0,Y 145.557,Z 263.099,A -85,B 0,C 180,E1 -28306.404,E2 -28306.404} C_VEL
LIN {X 0,Y 148.547,Z 271.039,A -85,B 0,C 180,E1 -28310.914,E2 -28310.914} C_VEL
LIN {X 0,Y 152.885,Z 278.737,A -85,B 0,C 180,E1 -28315.835,E2 -28315.835} C_VEL
LIN {X 0,Y 157.556,Z 284.501,A -85,B 0,C 180,E1 -28319.913,E2 -28319.913} C_VEL
LIN {X 0,Y 164.37,Z 290.622,A -85,B 0,C 180,E1 -28324.687,E2 -28324.687} C_VEL
LIN {X 0,Y 172.811,Z 295.905,A -85,B 0,C 180,E1 -28329.286,E2 -28329.286} C_VEL
LIN {X 0,Y 183.059,Z 300.42,A -85,B 0,C 180,E1 -28333.694,E2 -28333.694} C_VEL
LIN {X 0,Y 194.303,Z 303.895,A -85,B 0,C 180,E1 -28337.574,E2 -28337.574} C_VEL
LIN {X 0,Y 206.315,Z 306.532,A -85,B 0,C 180,E1 -28341.059,E2 -28341.059} C_VEL
LIN {X 0,Y 212.539,Z 307.623,A -85,B 0,C 180,E1 -28342.742,E2 -28342.742} C_VEL
LIN {X 0,Y 219.058,Z 308.523,A -85,B 0,C 180,E1 -28344.477,E2 -28344.477} C_VEL
LIN {X 0,Y 225.754,Z 309.356,A -85,B 0,C 180,E1 -28346.43,E2 -28346.43} C_VEL
LIN {X 0,Y 230.606,Z 309.805,A -85,B 0,C 180,E1 -28348.254,E2 -28348.254} C_VEL
LIN {X 0,Y 231.966,Z 309.881,A -85,B 0,C 180,E1 -28348.851,E2 -28348.851} C_VEL
LIN {X 0,Y 233.773,Z 309.904,A -85,B 0,C 180,E1 -28350,E2 -28350} C_VEL
LIN {X 0,Y 231.966,Z 309.881,A -85,B 0,C 180,E1 -28351.147,E2 -28351.147} C_VEL
LIN {X 0,Y 230.603,Z 309.805,A -85,B 0,C 180,E1 -28351.746,E2 -28351.746} C_VEL
LIN {X 0,Y 225.357,Z 309.316,A -85,B 0,C 180,E1 -28353.684,E2 -28353.684} C_VEL
LIN {X 0,Y 218.89,Z 308.513,A -85,B 0,C 180,E1 -28355.551,E2 -28355.551} C_VEL
LIN {X 0,Y 210.977,Z 307.389,A -85,B 0,C 180,E1 -28357.657,E2 -28357.657} C_VEL
LIN {X 0,Y 200.228,Z 305.329,A -85,B 0,C 180,E1 -28360.649,E2 -28360.649} C_VEL
LIN {X 0,Y 185.574,Z 301.302,A -85,B 0,C 180,E1 -28365.373,E2 -28365.373} C_VEL
LIN {X 0,Y 175.245,Z 297.176,A -85,B 0,C 180,E1 -28369.539,E2 -28369.539} C_VEL
LIN {X 0,Y 168.117,Z 293.252,A -85,B 0,C 180,E1 -28373.122,E2 -28373.122} C_VEL
LIN {X 0,Y 159.778,Z 286.733,A -85,B 0,C 180,E1 -28378.394,E2 -28378.394} C_VEL
LIN {X 0,Y 153.864,Z 280.084,A -85,B 0,C 180,E1 -28383.238,E2 -28383.238} C_VEL
LIN {X 0,Y 149.699,Z 273.448,A -85,B 0,C 180,E1 -28387.612,E2 -28387.612} C_VEL
LIN {X 0,Y 146.954,Z 267.288,A -85,B 0,C 180,E1 -28391.313,E2 -28391.313} C_VEL
LIN {X 0,Y 144.291,Z 258.317,A -85,B 0,C 180,E1 -28396.049,E2 -28396.049} C_VEL
LIN {X 0,Y 142.619,Z 249.391,A -85,B 0,C 180,E1 -28400.164,E2 -28400.164} C_VEL
LIN {X 0,Y 141.518,Z 241.573,A -85,B 0,C 180,E1 -28403.422,E2 -28403.422} C_VEL
LIN {X 0,Y 140.462,Z 231.29,A -85,B 0,C 180,E1 -28407.123,E2 -28407.123} C_VEL
LIN {X 0,Y 139.446,Z 220.634,A -85,B 0,C 180,E1 -28410.466,E2 -28410.466} C_VEL
LIN {X 0,Y 138.051,Z 212.479,A -85,B 0,C 180,E1 -28413.244,E2 -28413.244} C_VEL
LIN {X 0,Y 136.061,Z 205.713,A -85,B 0,C 180,E1 -28416.101,E2 -28416.101} C_VEL
LIN {X 0,Y 133.514,Z 198.797,A -85,B 0,C 180,E1 -28419.793,E2 -28419.793} C_VEL
LIN {X 0,Y 131.276,Z 193.431,A -85,B 0,C 180,E1 -28423.678,E2 -28423.678} C_VEL
LIN {X 0,Y 129.64,Z 189.946,A -85,B 0,C 180,E1 -28427.245,E2 -28427.245} C_VEL
LIN {X 0,Y 128.412,Z 187.135,A -85,B 0,C 180,E1 -28430.949,E2 -28430.949} C_VEL
LIN {X 0,Y 127.355,Z 183.317,A -85,B 0,C 180,E1 -28439.211,E2 -28439.211} C_VEL
LIN {X 0,Y 127.364,Z 183.488,A -85,B 0,C 180,E1 -28441.187,E2 -28441.187} C_VEL
LIN {X 0,Y 128.694,Z 187.717,A -85,B 0,C 180,E1 -28449.633,E2 -28449.633} C_VEL
LIN {X 0,Y 130.355,Z 191.516,A -85,B 0,C 180,E1 -28454.067,E2 -28454.067} C_VEL
LIN {X 0,Y 132.279,Z 195.762,A -85,B 0,C 180,E1 -28457.79,E2 -28457.79} C_VEL
LIN {X 0,Y 133.531,Z 199.166,A -85,B 0,C 180,E1 -28459.907,E2 -28459.907} C_VEL
LIN {X 0,Y 134.434,Z 202.89,A -85,B 0,C 180,E1 -28461.468,E2 -28461.468} C_VEL
LIN {X 0,Y 132.435,Z 218.348,A -85,B 0,C 180,E1 -28462.105,E2 -28462.105} C_VEL
LIN {X 0,Y 129.595,Z 230.259,A -85,B 0,C 180,E1 -28462.792,E2 -28462.792} C_VEL
LIN {X 0,Y 126.441,Z 240.026,A -85,B 0,C 180,E1 -28463.558,E2 -28463.558} C_VEL
LIN {X 0,Y 122.629,Z 249.401,A -85,B 0,C 180,E1 -28464.521,E2 -28464.521} C_VEL
LIN {X 0,Y 118.072,Z 258.671,A -85,B 0,C 180,E1 -28465.805,E2 -28465.805} C_VEL
LIN {X 0,Y 112.827,Z 267.608,A -85,B 0,C 180,E1 -28467.423,E2 -28467.423} C_VEL
LIN {X 0,Y 106.98,Z 276.13,A -85,B 0,C 180,E1 -28469.49,E2 -28469.49} C_VEL
LIN {X 0,Y 101.308,Z 283.343,A -85,B 0,C 180,E1 -28471.809,E2 -28471.809} C_VEL
LIN {X 0,Y 95.86,Z 289.541,A -85,B 0,C 180,E1 -28474.433,E2 -28474.433} C_VEL
LIN {X 0,Y 89.348,Z 296.074,A -85,B 0,C 180,E1 -28478.133,E2 -28478.133} C_VEL
LIN {X 0,Y 83.858,Z 301.143,A -85,B 0,C 180,E1 -28482.106,E2 -28482.106} C_VEL
LIN {X 0,Y 77.924,Z 306.071,A -85,B 0,C 180,E1 -28487.435,E2 -28487.435} C_VEL
LIN {X 0,Y 72.153,Z 310.397,A -85,B 0,C 180,E1 -28494.238,E2 -28494.238} C_VEL
LIN {X 0,Y 68.899,Z 312.766,A -85,B 0,C 180,E1 -28499.335,E2 -28499.335} C_VEL
LIN {X 0,Y 64.445,Z 315.969,A -85,B 0,C 180,E1 -28510.903,E2 -28510.903} C_VEL
LIN {X 0,Y 63.183,Z 317.036,A -85,B 0,C 180,E1 -28517.146,E2 -28517.146} C_VEL
LIN {X 0,Y 62.574,Z 317.635,A -85,B 0,C 180,E1 -28523.551,E2 -28523.551} C_VEL
LIN {X 0,Y 62.569,Z 317.798,A -85,B 0,C 180,E1 -28530,E2 -28530} C_VEL
LIN {X 0,Y 62.556,Z 317.635,A -85,B 0,C 180,E1 -28536.451,E2 -28536.451} C_VEL
LIN {X 0,Y 63.159,Z 317.036,A -85,B 0,C 180,E1 -28542.859,E2 -28542.859} C_VEL
LIN {X 0,Y 66.336,Z 314.572,A -85,B 0,C 180,E1 -28555.074,E2 -28555.074} C_VEL
LIN {X 0,Y 70.475,Z 311.615,A -85,B 0,C 180,E1 -28563.262,E2 -28563.262} C_VEL
LIN {X 0,Y 75.848,Z 307.623,A -85,B 0,C 180,E1 -28570.437,E2 -28570.437} C_VEL
LIN {X 0,Y 81.474,Z 303.194,A -85,B 0,C 180,E1 -28575.846,E2 -28575.846} C_VEL
LIN {X 0,Y 88.164,Z 297.232,A -85,B 0,C 180,E1 -28581.007,E2 -28581.007} C_VEL
LIN {X 0,Y 94.534,Z 290.916,A -85,B 0,C 180,E1 -28584.863,E2 -28584.863} C_VEL
LIN {X 0,Y 99.942,Z 284.969,A -85,B 0,C 180,E1 -28587.548,E2 -28587.548} C_VEL
LIN {X 0,Y 105.561,Z 278.048,A -85,B 0,C 180,E1 -28589.94,E2 -28589.94} C_VEL
LIN {X 0,Y 111.362,Z 269.876,A -85,B 0,C 180,E1 -28592.071,E2 -28592.071} C_VEL
LIN {X 0,Y 116.563,Z 261.371,A -85,B 0,C 180,E1 -28593.748,E2 -28593.748} C_VEL
LIN {X 0,Y 121.102,Z 252.662,A -85,B 0,C 180,E1 -28595.063,E2 -28595.063} C_VEL
LIN {X 0,Y 124.937,Z 243.985,A -85,B 0,C 180,E1 -28596.045,E2 -28596.045} C_VEL
LIN {X 0,Y 128.546,Z 233.726,A -85,B 0,C 180,E1 -28596.96,E2 -28596.96} C_VEL
LIN {X 0,Y 131.261,Z 223.593,A -85,B 0,C 180,E1 -28597.631,E2 -28597.631} C_VEL
LIN {X 0,Y 133.143,Z 213.745,A -85,B 0,C 180,E1 -28598.09,E2 -28598.09} C_VEL
LIN {X 0,Y 134.434,Z 202.892,A -85,B 0,C 180,E1 -28598.532,E2 -28598.532} C_VEL
LIN {X 0,Y 133.155,Z 197.918,A -85,B 0,C 180,E1 -28600.737,E2 -28600.737} C_VEL
LIN {X 0,Y 131.072,Z 193.022,A -85,B 0,C 180,E1 -28604.447,E2 -28604.447} C_VEL
LIN {X 0,Y 129.541,Z 189.738,A -85,B 0,C 180,E1 -28607.872,E2 -28607.872} C_VEL
LIN {X 0,Y 128.53,Z 187.257,A -85,B 0,C 180,E1 -28610.954,E2 -28610.954} C_VEL
LIN {X 0,Y 127.36,Z 183.374,A -85,B 0,C 180,E1 -28619.208,E2 -28619.208} C_VEL
LIN {X 0,Y 127.364,Z 183.583,A -85,B 0,C 180,E1 -28621.777,E2 -28621.777} C_VEL
LIN {X 0,Y 128.715,Z 187.721,A -85,B 0,C 180,E1 -28630.067,E2 -28630.067} C_VEL
LIN {X 0,Y 130.343,Z 191.516,A -85,B 0,C 180,E1 -28634.424,E2 -28634.424} C_VEL
LIN {X 0,Y 132.342,Z 195.913,A -85,B 0,C 180,E1 -28638.278,E2 -28638.278} C_VEL
LIN {X 0,Y 134.913,Z 202.433,A -85,B 0,C 180,E1 -28642.289,E2 -28642.289} C_VEL
LIN {X 0,Y 137.342,Z 209.933,A -85,B 0,C 180,E1 -28645.781,E2 -28645.781} C_VEL
LIN {X 0,Y 138.829,Z 216.313,A -85,B 0,C 180,E1 -28648.125,E2 -28648.125} C_VEL
LIN {X 0,Y 139.955,Z 225.157,A -85,B 0,C 180,E1 -28650.893,E2 -28650.893} C_VEL
LIN {X 0,Y 140.997,Z 236.728,A -85,B 0,C 180,E1 -28654.78,E2 -28654.78} C_VEL
LIN {X 0,Y 141.983,Z 245.458,A -85,B 0,C 180,E1 -28658.127,E2 -28658.127} C_VEL
LIN {X 0,Y 142.215,Z 249.812,A -85,B 0,C 180,E1 -28659.755,E2 -28659.755} C_VEL
LIN {X 0,Y 141.052,Z 257.577,A -85,B 0,C 180,E1 -28662.222,E2 -28662.222} C_VEL
LIN {X 0,Y 139.978,Z 264.913,A -85,B 0,C 180,E1 -28664.875,E2 -28664.875} C_VEL
LIN {X 0,Y 140.289,Z 268.597,A -85,B 0,C 180,E1 -28666.735,E2 -28666.735} C_VEL
LIN {X 0,Y 143.888,Z 277.516,A -85,B 0,C 180,E1 -28672.53,E2 -28672.53} C_VEL
LIN {X 0,Y 148.928,Z 285.062,A -85,B 0,C 180,E1 -28678.147,E2 -28678.147} C_VEL
LIN {X 0,Y 154.802,Z 290.902,A -85,B 0,C 180,E1 -28683,E2 -28683} C_VEL
LIN {X 0,Y 162.802,Z 296.462,A -85,B 0,C 180,E1 -28688.142,E2 -28688.142} C_VEL
LIN {X 0,Y 170.157,Z 300.016,A -85,B 0,C 180,E1 -28691.795,E2 -28691.795} C_VEL
LIN {X 0,Y 182.213,Z 304.1,A -85,B 0,C 180,E1 -28696.619,E2 -28696.619} C_VEL
LIN {X 0,Y 192.691,Z 306.524,A -85,B 0,C 180,E1 -28699.98,E2 -28699.98} C_VEL
LIN {X 0,Y 205.148,Z 308.503,A -85,B 0,C 180,E1 -28703.447,E2 -28703.447} C_VEL
LIN {X 0,Y 215.64,Z 309.63,A -85,B 0,C 180,E1 -28706.263,E2 -28706.263} C_VEL
LIN {X 0,Y 221.846,Z 310.039,A -85,B 0,C 180,E1 -28708.185,E2 -28708.185} C_VEL
LIN {X 0,Y 224.907,Z 310.12,A -85,B 0,C 180,E1 -28709.333,E2 -28709.333} C_VEL
LIN {X 0,Y 226.133,Z 310.105,A -85,B 0,C 180,E1 -28710,E2 -28710} C_VEL
LIN {X 0,Y 224.907,Z 310.12,A -85,B 0,C 180,E1 -28710.666,E2 -28710.666} C_VEL
LIN {X 0,Y 221.842,Z 310.039,A -85,B 0,C 180,E1 -28711.815,E2 -28711.815} C_VEL
LIN {X 0,Y 215.576,Z 309.632,A -85,B 0,C 180,E1 -28713.738,E2 -28713.738} C_VEL
LIN {X 0,Y 207.848,Z 308.821,A -85,B 0,C 180,E1 -28715.822,E2 -28715.822} C_VEL
LIN {X 0,Y 198.84,Z 307.609,A -85,B 0,C 180,E1 -28718.254,E2 -28718.254} C_VEL
LIN {X 0,Y 186.709,Z 305.261,A -85,B 0,C 180,E1 -28721.859,E2 -28721.859} C_VEL
LIN {X 0,Y 174.305,Z 301.61,A -85,B 0,C 180,E1 -28726.394,E2 -28726.394} C_VEL
LIN {X 0,Y 165.163,Z 297.738,A -85,B 0,C 180,E1 -28730.59,E2 -28730.59} C_VEL
LIN {X 0,Y 158.363,Z 293.669,A -85,B 0,C 180,E1 -28734.553,E2 -28734.553} C_VEL
LIN {X 0,Y 152.42,Z 288.84,A -85,B 0,C 180,E1 -28738.83,E2 -28738.83} C_VEL
LIN {X 0,Y 146.604,Z 282.027,A -85,B 0,C 180,E1 -28744.217,E2 -28744.217} C_VEL
LIN {X 0,Y 142.673,Z 275.042,A -85,B 0,C 180,E1 -28749.16,E2 -28749.16} C_VEL
LIN {X 0,Y 139.784,Z 266.905,A -85,B 0,C 180,E1 -28754.242,E2 -28754.242} C_VEL
LIN {X 0,Y 138.15,Z 258.938,A -85,B 0,C 180,E1 -28758.6,E2 -28758.6} C_VEL
LIN {X 0,Y 137.074,Z 249.818,A -85,B 0,C 180,E1 -28762.958,E2 -28762.958} C_VEL
LIN {X 0,Y 136.488,Z 241.221,A -85,B 0,C 180,E1 -28766.57,E2 -28766.57} C_VEL
LIN {X 0,Y 136.015,Z 230.972,A -85,B 0,C 180,E1 -28770.306,E2 -28770.306} C_VEL
LIN {X 0,Y 135.517,Z 221.763,A -85,B 0,C 180,E1 -28773.328,E2 -28773.328} C_VEL
LIN {X 0,Y 134.435,Z 214.604,A -85,B 0,C 180,E1 -28776.101,E2 -28776.101} C_VEL
LIN {X 0,Y 132.353,Z 207.144,A -85,B 0,C 180,E1 -28779.811,E2 -28779.811} C_VEL
LIN {X 0,Y 130.472,Z 201.834,A -85,B 0,C 180,E1 -28783.273,E2 -28783.273} C_VEL
LIN {X 0,Y 128.574,Z 197.049,A -85,B 0,C 180,E1 -28787.593,E2 -28787.593} C_VEL
LIN {X 0,Y 127.274,Z 193.867,A -85,B 0,C 180,E1 -28791.867,E2 -28791.867} C_VEL
LIN {X 0,Y 126.486,Z 190.394,A -85,B 0,C 180,E1 -28799.206,E2 -28799.206} C_VEL
LIN {X 0,Y 126.484,Z 190.542,A -85,B 0,C 180,E1 -28800.897,E2 -28800.897} C_VEL
LIN {X 0,Y 127.57,Z 194.593,A -85,B 0,C 180,E1 -28808.915,E2 -28808.915} C_VEL
LIN {X 0,Y 129.006,Z 198.217,A -85,B 0,C 180,E1 -28813.165,E2 -28813.165} C_VEL
LIN {X 0,Y 130.562,Z 202.024,A -85,B 0,C 180,E1 -28816.518,E2 -28816.518} C_VEL
LIN {X 0,Y 131.436,Z 204.745,A -85,B 0,C 180,E1 -28818.21,E2 -28818.21} C_VEL
LIN {X 0,Y 131.669,Z 205.752,A -85,B 0,C 180,E1 -28818.68,E2 -28818.68} C_VEL
LIN {X 0,Y 129.63,Z 219.494,A -85,B 0,C 180,E1 -28819.272,E2 -28819.272} C_VEL
LIN {X 0,Y 127.013,Z 230.069,A -85,B 0,C 180,E1 -28819.838,E2 -28819.838} C_VEL
LIN {X 0,Y 123.593,Z 240.299,A -85,B 0,C 180,E1 -28820.586,E2 -28820.586} C_VEL
LIN {X 0,Y 119.075,Z 250.841,A -85,B 0,C 180,E1 -28821.629,E2 -28821.629} C_VEL
LIN {X 0,Y 114.377,Z 259.83,A -85,B 0,C 180,E1 -28822.827,E2 -28822.827} C_VEL
LIN {X 0,Y 108.981,Z 268.552,A -85,B 0,C 180,E1 -28824.371,E2 -28824.371} C_VEL
LIN {X 0,Y 103.665,Z 275.939,A -85,B 0,C 180,E1 -28826.066,E2 -28826.066} C_VEL
LIN {X 0,Y 97.738,Z 283.152,A -85,B 0,C 180,E1 -28828.255,E2 -28828.255} C_VEL
LIN {X 0,Y 92.028,Z 289.35,A -85,B 0,C 180,E1 -28830.78,E2 -28830.78} C_VEL
LIN {X 0,Y 85.134,Z 295.883,A -85,B 0,C 180,E1 -28834.359,E2 -28834.359} C_VEL
LIN {X 0,Y 78.592,Z 301.457,A -85,B 0,C 180,E1 -28838.757,E2 -28838.757} C_VEL
LIN {X 0,Y 72.843,Z 305.88,A -85,B 0,C 180,E1 -28843.647,E2 -28843.647} C_VEL
LIN {X 0,Y 66.508,Z 310.206,A -85,B 0,C 180,E1 -28850.653,E2 -28850.653} C_VEL
LIN {X 0,Y 62.883,Z 312.575,A -85,B 0,C 180,E1 -28856.026,E2 -28856.026} C_VEL
LIN {X 0,Y 57.739,Z 315.777,A -85,B 0,C 180,E1 -28868.582,E2 -28868.582} C_VEL
LIN {X 0,Y 56.27,Z 316.846,A -85,B 0,C 180,E1 -28875.535,E2 -28875.535} C_VEL
LIN {X 0,Y 55.528,Z 317.445,A -85,B 0,C 180,E1 -28882.729,E2 -28882.729} C_VEL
LIN {X 0,Y 55.48,Z 317.608,A -85,B 0,C 180,E1 -28890,E2 -28890} C_VEL
LIN {X 0,Y 55.491,Z 317.444,A -85,B 0,C 180,E1 -28897.276,E2 -28897.276} C_VEL
LIN {X 0,Y 56.251,Z 316.845,A -85,B 0,C 180,E1 -28904.47,E2 -28904.47} C_VEL
LIN {X 0,Y 59.938,Z 314.38,A -85,B 0,C 180,E1 -28917.97,E2 -28917.97} C_VEL
LIN {X 0,Y 64.645,Z 311.424,A -85,B 0,C 180,E1 -28926.722,E2 -28926.722} C_VEL
LIN {X 0,Y 70.581,Z 307.432,A -85,B 0,C 180,E1 -28934.188,E2 -28934.188} C_VEL
LIN {X 0,Y 77.518,Z 302.318,A -85,B 0,C 180,E1 -28940.379,E2 -28940.379} C_VEL
LIN {X 0,Y 83.848,Z 297.04,A -85,B 0,C 180,E1 -28944.808,E2 -28944.808} C_VEL
LIN {X 0,Y 90.618,Z 290.725,A -85,B 0,C 180,E1 -28948.553,E2 -28948.553} C_VEL
LIN {X 0,Y 96.308,Z 284.778,A -85,B 0,C 180,E1 -28951.126,E2 -28951.126} C_VEL
LIN {X 0,Y 102.181,Z 277.857,A -85,B 0,C 180,E1 -28953.398,E2 -28953.398} C_VEL
LIN {X 0,Y 108.219,Z 269.686,A -85,B 0,C 180,E1 -28955.393,E2 -28955.393} C_VEL
LIN {X 0,Y 113.597,Z 261.18,A -85,B 0,C 180,E1 -28956.967,E2 -28956.967} C_VEL
LIN {X 0,Y 118.29,Z 252.472,A -85,B 0,C 180,E1 -28958.176,E2 -28958.176} C_VEL
LIN {X 0,Y 122.136,Z 244.026,A -85,B 0,C 180,E1 -28959.067,E2 -28959.067} C_VEL
LIN {X 0,Y 125.593,Z 234.677,A -85,B 0,C 180,E1 -28959.847,E2 -28959.847} C_VEL
LIN {X 0,Y 128.61,Z 223.926,A -85,B 0,C 180,E1 -28960.525,E2 -28960.525} C_VEL
LIN {X 0,Y 130.687,Z 213.386,A -85,B 0,C 180,E1 -28960.983,E2 -28960.983} C_VEL
LIN {X 0,Y 131.67,Z 205.743,A -85,B 0,C 180,E1 -28961.32,E2 -28961.32} C_VEL
LIN {X 0,Y 130.899,Z 202.994,A -85,B 0,C 180,E1 -28962.823,E2 -28962.823} C_VEL
LIN {X 0,Y 129.252,Z 198.818,A -85,B 0,C 180,E1 -28966.247,E2 -28966.247} C_VEL
LIN {X 0,Y 128.228,Z 196.292,A -85,B 0,C 180,E1 -28968.918,E2 -28968.918} C_VEL
LIN {X 0,Y 127.318,Z 193.965,A -85,B 0,C 180,E1 -28972.066,E2 -28972.066} C_VEL
LIN {X 0,Y 126.492,Z 190.293,A -85,B 0,C 180,E1 -28979.998,E2 -28979.998} C_VEL
LIN {X 0,Y 126.474,Z 190.998,A -85,B 0,C 180,E1 -28982.088,E2 -28982.088} C_VEL
LIN {X 0,Y 127.578,Z 194.588,A -85,B 0,C 180,E1 -28989.313,E2 -28989.313} C_VEL
LIN {X 0,Y 129.062,Z 198.363,A -85,B 0,C 180,E1 -28993.68,E2 -28993.68} C_VEL
LIN {X 0,Y 130.762,Z 202.617,A -85,B 0,C 180,E1 -28997.293,E2 -28997.293} C_VEL
LIN {X 0,Y 132.628,Z 208.148,A -85,B 0,C 180,E1 -29000.753,E2 -29000.753} C_VEL
LIN {X 0,Y 134.572,Z 215.257,A -85,B 0,C 180,E1 -29004.18,E2 -29004.18} C_VEL
LIN {X 0,Y 135.507,Z 221.806,A -85,B 0,C 180,E1 -29006.675,E2 -29006.675} C_VEL
LIN {X 0,Y 135.97,Z 229.551,A -85,B 0,C 180,E1 -29009.237,E2 -29009.237} C_VEL
LIN {X 0,Y 136.364,Z 238.486,A -85,B 0,C 180,E1 -29012.408,E2 -29012.408} C_VEL
LIN {X 0,Y 136.731,Z 245.934,A -85,B 0,C 180,E1 -29015.324,E2 -29015.324} C_VEL
LIN {X 0,Y 137.638,Z 255.459,A -85,B 0,C 180,E1 -29019.662,E2 -29019.662} C_VEL
LIN {X 0,Y 139.084,Z 263.932,A -85,B 0,C 180,E1 -29024.085,E2 -29024.085} C_VEL
LIN {X 0,Y 140.289,Z 268.597,A -85,B 0,C 180,E1 -29026.735,E2 -29026.735} C_VEL
LIN {X 0,Y 140.724,Z 272.15,A -85,B 0,C 180,E1 -29028.684,E2 -29028.684} C_VEL
LIN {X 0,Y 140.175,Z 278.485,A -85,B 0,C 180,E1 -29031.844,E2 -29031.844} C_VEL
LIN {X 0,Y 140.157,Z 284.173,A -85,B 0,C 180,E1 -29035.123,E2 -29035.123} C_VEL
LIN {X 0,Y 141.407,Z 286.763,A -85,B 0,C 180,E1 -29037.165,E2 -29037.165} C_VEL
LIN {X 0,Y 146.847,Z 292.423,A -85,B 0,C 180,E1 -29042.294,E2 -29042.294} C_VEL
LIN {X 0,Y 154.718,Z 297.922,A -85,B 0,C 180,E1 -29047.865,E2 -29047.865} C_VEL
LIN {X 0,Y 163.338,Z 301.912,A -85,B 0,C 180,E1 -29052.471,E2 -29052.471} C_VEL
LIN {X 0,Y 173.329,Z 305.097,A -85,B 0,C 180,E1 -29056.683,E2 -29056.683} C_VEL
LIN {X 0,Y 187.544,Z 308.018,A -85,B 0,C 180,E1 -29061.379,E2 -29061.379} C_VEL
LIN {X 0,Y 197.782,Z 309.285,A -85,B 0,C 180,E1 -29064.228,E2 -29064.228} C_VEL
LIN {X 0,Y 204.809,Z 309.923,A -85,B 0,C 180,E1 -29066.065,E2 -29066.065} C_VEL
LIN {X 0,Y 212.372,Z 310.292,A -85,B 0,C 180,E1 -29068.104,E2 -29068.104} C_VEL
LIN {X 0,Y 218.041,Z 310.318,A -85,B 0,C 180,E1 -29070,E2 -29070} C_VEL
LIN {X 0,Y 211.001,Z 310.233,A -85,B 0,C 180,E1 -29072.27,E2 -29072.27} C_VEL
LIN {X 0,Y 204.32,Z 309.888,A -85,B 0,C 180,E1 -29074.059,E2 -29074.059} C_VEL
LIN {X 0,Y 187.483,Z 308.019,A -85,B 0,C 180,E1 -29078.624,E2 -29078.624} C_VEL
LIN {X 0,Y 173.328,Z 305.098,A -85,B 0,C 180,E1 -29083.316,E2 -29083.316} C_VEL
LIN {X 0,Y 162.479,Z 301.613,A -85,B 0,C 180,E1 -29087.902,E2 -29087.902} C_VEL
LIN {X 0,Y 154.72,Z 297.922,A -85,B 0,C 180,E1 -29092.135,E2 -29092.135} C_VEL
LIN {X 0,Y 146.846,Z 292.424,A -85,B 0,C 180,E1 -29097.705,E2 -29097.705} C_VEL
LIN {X 0,Y 141.031,Z 286.292,A -85,B 0,C 180,E1 -29103.241,E2 -29103.241} C_VEL
LIN {X 0,Y 137.184,Z 280.022,A -85,B 0,C 180,E1 -29108.291,E2 -29108.291} C_VEL
LIN {X 0,Y 134.665,Z 273.354,A -85,B 0,C 180,E1 -29113.062,E2 -29113.062} C_VEL
LIN {X 0,Y 133.113,Z 266.071,A -85,B 0,C 180,E1 -29117.66,E2 -29117.66} C_VEL
LIN {X 0,Y 132.335,Z 258.875,A -85,B 0,C 180,E1 -29121.685,E2 -29121.685} C_VEL
LIN {X 0,Y 131.958,Z 250.215,A -85,B 0,C 180,E1 -29125.942,E2 -29125.942} C_VEL
LIN {X 0,Y 131.952,Z 240.368,A -85,B 0,C 180,E1 -29130.101,E2 -29130.101} C_VEL
LIN {X 0,Y 132.091,Z 231.667,A -85,B 0,C 180,E1 -29133.285,E2 -29133.285} C_VEL
LIN {X 0,Y 131.903,Z 223.454,A -85,B 0,C 180,E1 -29136.24,E2 -29136.24} C_VEL
LIN {X 0,Y 131.007,Z 217.068,A -85,B 0,C 180,E1 -29139.081,E2 -29139.081} C_VEL
LIN {X 0,Y 129.607,Z 210.958,A -85,B 0,C 180,E1 -29142.548,E2 -29142.548} C_VEL
LIN {X 0,Y 128.129,Z 206.064,A -85,B 0,C 180,E1 -29146.218,E2 -29146.218} C_VEL
LIN {X 0,Y 126.825,Z 202.594,A -85,B 0,C 180,E1 -29150.029,E2 -29150.029} C_VEL
LIN {X 0,Y 126.255,Z 200.797,A -85,B 0,C 180,E1 -29152.405,E2 -29152.405} C_VEL
LIN {X 0,Y 125.628,Z 197.331,A -85,B 0,C 180,E1 -29160.002,E2 -29160.002} C_VEL
LIN {X 0,Y 126.47,Z 201.46,A -85,B 0,C 180,E1 -29168.188,E2 -29168.188} C_VEL
LIN {X 0,Y 127.756,Z 205.048,A -85,B 0,C 180,E1 -29172.411,E2 -29172.411} C_VEL
LIN {X 0,Y 129.147,Z 209.179,A -85,B 0,C 180,E1 -29175.844,E2 -29175.844} C_VEL
LIN {X 0,Y 127.179,Z 220.547,A -85,B 0,C 180,E1 -29176.321,E2 -29176.321} C_VEL
LIN {X 0,Y 124.779,Z 229.878,A -85,B 0,C 180,E1 -29176.765,E2 -29176.765} C_VEL
LIN {X 0,Y 121.06,Z 240.651,A -85,B 0,C 180,E1 -29177.488,E2 -29177.488} C_VEL
LIN {X 0,Y 116.646,Z 250.651,A -85,B 0,C 180,E1 -29178.387,E2 -29178.387} C_VEL
LIN {X 0,Y 111.817,Z 259.64,A -85,B 0,C 180,E1 -29179.475,E2 -29179.475} C_VEL
LIN {X 0,Y 106.241,Z 268.361,A -85,B 0,C 180,E1 -29180.87,E2 -29180.87} C_VEL
LIN {X 0,Y 100.737,Z 275.748,A -85,B 0,C 180,E1 -29182.423,E2 -29182.423} C_VEL
LIN {X 0,Y 94.579,Z 282.961,A -85,B 0,C 180,E1 -29184.457,E2 -29184.457} C_VEL
LIN {X 0,Y 88.59,Z 289.159,A -85,B 0,C 180,E1 -29186.814,E2 -29186.814} C_VEL
LIN {X 0,Y 81.324,Z 295.691,A -85,B 0,C 180,E1 -29190.209,E2 -29190.209} C_VEL
LIN {X 0,Y 73.757,Z 301.689,A -85,B 0,C 180,E1 -29194.874,E2 -29194.874} C_VEL
LIN {X 0,Y 68.127,Z 305.689,A -85,B 0,C 180,E1 -29199.312,E2 -29199.312} C_VEL
LIN {X 0,Y 61.172,Z 310.015,A -85,B 0,C 180,E1 -29206.422,E2 -29206.422} C_VEL
LIN {X 0,Y 57.125,Z 312.384,A -85,B 0,C 180,E1 -29212.038,E2 -29212.038} C_VEL
LIN {X 0,Y 53.734,Z 314.188,A -85,B 0,C 180,E1 -29218.455,E2 -29218.455} C_VEL
LIN {X 0,Y 49.391,Z 316.654,A -85,B 0,C 180,E1 -29233.466,E2 -29233.466} C_VEL
LIN {X 0,Y 48.486,Z 317.254,A -85,B 0,C 180,E1 -29241.666,E2 -29241.666} C_VEL
LIN {X 0,Y 48.375,Z 317.417,A -85,B 0,C 180,E1 -29250,E2 -29250} C_VEL
LIN {X 0,Y 48.437,Z 317.253,A -85,B 0,C 180,E1 -29258.343,E2 -29258.343} C_VEL
LIN {X 0,Y 49.375,Z 316.654,A -85,B 0,C 180,E1 -29266.539,E2 -29266.539} C_VEL
LIN {X 0,Y 53.734,Z 314.188,A -85,B 0,C 180,E1 -29281.545,E2 -29281.545} C_VEL
LIN {X 0,Y 59.077,Z 311.233,A -85,B 0,C 180,E1 -29290.866,E2 -29290.866} C_VEL
LIN {X 0,Y 65.666,Z 307.241,A -85,B 0,C 180,E1 -29298.519,E2 -29298.519} C_VEL
LIN {X 0,Y 72.452,Z 302.652,A -85,B 0,C 180,E1 -29304.177,E2 -29304.177} C_VEL
LIN {X 0,Y 79.949,Z 296.848,A -85,B 0,C 180,E1 -29308.99,E2 -29308.99} C_VEL
LIN {X 0,Y 87.119,Z 290.534,A -85,B 0,C 180,E1 -29312.546,E2 -29312.546} C_VEL
LIN {X 0,Y 93.083,Z 284.588,A -85,B 0,C 180,E1 -29314.962,E2 -29314.962} C_VEL
LIN {X 0,Y 99.198,Z 277.666,A -85,B 0,C 180,E1 -29317.076,E2 -29317.076} C_VEL
LIN {X 0,Y 105.456,Z 269.495,A -85,B 0,C 180,E1 -29318.909,E2 -29318.909} C_VEL
LIN {X 0,Y 111.012,Z 260.99,A -85,B 0,C 180,E1 -29320.341,E2 -29320.341} C_VEL
LIN {X 0,Y 115.842,Z 252.282,A -85,B 0,C 180,E1 -29321.433,E2 -29321.433} C_VEL
LIN {X 0,Y 119.677,Z 244.108,A -85,B 0,C 180,E1 -29322.212,E2 -29322.212} C_VEL
LIN {X 0,Y 123.376,Z 234.329,A -85,B 0,C 180,E1 -29322.955,E2 -29322.955} C_VEL
LIN {X 0,Y 126.43,Z 223.696,A -85,B 0,C 180,E1 -29323.561,E2 -29323.561} C_VEL
LIN {X 0,Y 128.58,Z 212.995,A -85,B 0,C 180,E1 -29323.981,E2 -29323.981} C_VEL
LIN {X 0,Y 129.103,Z 209.11,A -85,B 0,C 180,E1 -29324.204,E2 -29324.204} C_VEL
LIN {X 0,Y 127.789,Z 205.175,A -85,B 0,C 180,E1 -29327.492,E2 -29327.492} C_VEL
LIN {X 0,Y 126.823,Z 202.546,A -85,B 0,C 180,E1 -29330.429,E2 -29330.429} C_VEL
LIN {X 0,Y 126.247,Z 200.812,A -85,B 0,C 180,E1 -29332.803,E2 -29332.803} C_VEL
LIN {X 0,Y 125.624,Z 197.364,A -85,B 0,C 180,E1 -29339.998,E2 -29339.998} C_VEL
LIN {X 0,Y 126.432,Z 201.302,A -85,B 0,C 180,E1 -29348.389,E2 -29348.389} C_VEL
LIN {X 0,Y 127.758,Z 205.124,A -85,B 0,C 180,E1 -29352.811,E2 -29352.811} C_VEL
LIN {X 0,Y 128.921,Z 208.728,A -85,B 0,C 180,E1 -29355.917,E2 -29355.917} C_VEL
LIN {X 0,Y 130.382,Z 214.009,A -85,B 0,C 180,E1 -29359.276,E2 -29359.276} C_VEL
LIN {X 0,Y 131.516,Z 220.357,A -85,B 0,C 180,E1 -29362.482,E2 -29362.482} C_VEL
LIN {X 0,Y 132.032,Z 225.069,A -85,B 0,C 180,E1 -29364.362,E2 -29364.362} C_VEL
LIN {X 0,Y 132.015,Z 237.03,A -85,B 0,C 180,E1 -29368.626,E2 -29368.626} C_VEL
LIN {X 0,Y 131.924,Z 246.003,A -85,B 0,C 180,E1 -29372.188,E2 -29372.188} C_VEL
LIN {X 0,Y 132.052,Z 254.048,A -85,B 0,C 180,E1 -29375.832,E2 -29375.832} C_VEL
LIN {X 0,Y 132.656,Z 262.78,A -85,B 0,C 180,E1 -29380.399,E2 -29380.399} C_VEL
LIN {X 0,Y 134.196,Z 271.635,A -85,B 0,C 180,E1 -29385.785,E2 -29385.785} C_VEL
LIN {X 0,Y 136.507,Z 278.496,A -85,B 0,C 180,E1 -29390.555,E2 -29390.555} C_VEL
LIN {X 0,Y 140.12,Z 285.06,A -85,B 0,C 180,E1 -29395.699,E2 -29395.699} C_VEL
LIN {X 0,Y 141.407,Z 286.763,A -85,B 0,C 180,E1 -29397.165,E2 -29397.165} C_VEL
LIN {X 0,Y 142.839,Z 289.45,A -85,B 0,C 180,E1 -29399.236,E2 -29399.236} C_VEL
LIN {X 0,Y 143.861,Z 294.027,A -85,B 0,C 180,E1 -29402.733,E2 -29402.733} C_VEL
LIN {X 0,Y 145.417,Z 298.084,A -85,B 0,C 180,E1 -29406.238,E2 -29406.238} C_VEL
LIN {X 0,Y 147.63,Z 299.906,A -85,B 0,C 180,E1 -29408.241,E2 -29408.241} C_VEL
LIN {X 0,Y 154.849,Z 303.142,A -85,B 0,C 180,E1 -29412.379,E2 -29412.379} C_VEL
LIN {X 0,Y 167.336,Z 306.786,A -85,B 0,C 180,E1 -29417.878,E2 -29417.878} C_VEL
LIN {X 0,Y 177.68,Z 308.653,A -85,B 0,C 180,E1 -29421.429,E2 -29421.429} C_VEL
LIN {X 0,Y 193.358,Z 310.232,A -85,B 0,C 180,E1 -29425.831,E2 -29425.831} C_VEL
LIN {X 0,Y 203.873,Z 310.626,A -85,B 0,C 180,E1 -29428.547,E2 -29428.547} C_VEL
LIN {X 0,Y 208.84,Z 310.56,A -85,B 0,C 180,E1 -29430,E2 -29430} C_VEL
LIN {X 0,Y 201.711,Z 310.577,A -85,B 0,C 180,E1 -29431.997,E2 -29431.997} C_VEL
LIN {X 0,Y 190.451,Z 310.041,A -85,B 0,C 180,E1 -29434.913,E2 -29434.913} C_VEL
LIN {X 0,Y 175.645,Z 308.335,A -85,B 0,C 180,E1 -29439.21,E2 -29439.21} C_VEL
LIN {X 0,Y 165.721,Z 306.418,A -85,B 0,C 180,E1 -29442.742,E2 -29442.742} C_VEL
LIN {X 0,Y 152.548,Z 302.212,A -85,B 0,C 180,E1 -29448.814,E2 -29448.814} C_VEL
LIN {X 0,Y 145.401,Z 298.586,A -85,B 0,C 180,E1 -29453.315,E2 -29453.315} C_VEL
LIN {X 0,Y 139.299,Z 294.248,A -85,B 0,C 180,E1 -29458.176,E2 -29458.176} C_VEL
LIN {X 0,Y 134.503,Z 289.169,A -85,B 0,C 180,E1 -29463.281,E2 -29463.281} C_VEL
LIN {X 0,Y 130.275,Z 281.775,A -85,B 0,C 180,E1 -29469.763,E2 -29469.763} C_VEL
LIN {X 0,Y 128.318,Z 275.549,A -85,B 0,C 180,E1 -29474.604,E2 -29474.604} C_VEL
LIN {X 0,Y 127.246,Z 268.102,A -85,B 0,C 180,E1 -29479.644,E2 -29479.644} C_VEL
LIN {X 0,Y 126.99,Z 259.83,A -85,B 0,C 180,E1 -29484.476,E2 -29484.476} C_VEL
LIN {X 0,Y 127.288,Z 250.055,A -85,B 0,C 180,E1 -29489.382,E2 -29489.382} C_VEL
LIN {X 0,Y 127.926,Z 240.625,A -85,B 0,C 180,E1 -29493.392,E2 -29493.392} C_VEL
LIN {X 0,Y 128.555,Z 231.122,A -85,B 0,C 180,E1 -29496.913,E2 -29496.913} C_VEL
LIN {X 0,Y 128.568,Z 226.007,A -85,B 0,C 180,E1 -29499.022,E2 -29499.022} C_VEL
LIN {X 0,Y 127.884,Z 219.968,A -85,B 0,C 180,E1 -29502.099,E2 -29502.099} C_VEL
LIN {X 0,Y 127.07,Z 214.951,A -85,B 0,C 180,E1 -29505.386,E2 -29505.386} C_VEL
LIN {X 0,Y 126.142,Z 211.361,A -85,B 0,C 180,E1 -29508.553,E2 -29508.553} C_VEL
LIN {X 0,Y 125.266,Z 208.021,A -85,B 0,C 180,E1 -29512.547,E2 -29512.547} C_VEL
LIN {X 0,Y 124.737,Z 204.588,A -85,B 0,C 180,E1 -29520.002,E2 -29520.002} C_VEL
LIN {X 0,Y 125.317,Z 208.158,A -85,B 0,C 180,E1 -29527.251,E2 -29527.251} C_VEL
LIN {X 0,Y 126.253,Z 211.504,A -85,B 0,C 180,E1 -29531.237,E2 -29531.237} C_VEL
LIN {X 0,Y 126.743,Z 213.332,A -85,B 0,C 180,E1 -29532.928,E2 -29532.928} C_VEL
LIN {X 0,Y 124.043,Z 225.909,A -85,B 0,C 180,E1 -29533.415,E2 -29533.415} C_VEL
LIN {X 0,Y 119.536,Z 239.485,A -85,B 0,C 180,E1 -29534.186,E2 -29534.186} C_VEL
LIN {X 0,Y 115.432,Z 248.829,A -85,B 0,C 180,E1 -29534.864,E2 -29534.864} C_VEL
LIN {X 0,Y 110.472,Z 258.099,A -85,B 0,C 180,E1 -29535.8,E2 -29535.8} C_VEL
LIN {X 0,Y 104.735,Z 267.037,A -85,B 0,C 180,E1 -29537.019,E2 -29537.019} C_VEL
LIN {X 0,Y 98.247,Z 275.557,A -85,B 0,C 180,E1 -29538.59,E2 -29538.59} C_VEL
LIN {X 0,Y 91.867,Z 282.77,A -85,B 0,C 180,E1 -29540.422,E2 -29540.422} C_VEL
LIN {X 0,Y 85.605,Z 288.967,A -85,B 0,C 180,E1 -29542.542,E2 -29542.542} C_VEL
LIN {X 0,Y 77.983,Z 295.5,A -85,B 0,C 180,E1 -29545.681,E2 -29545.681} C_VEL
LIN {X 0,Y 72.136,Z 300.003,A -85,B 0,C 180,E1 -29548.736,E2 -29548.736} C_VEL
LIN {X 0,Y 63.842,Z 305.497,A -85,B 0,C 180,E1 -29554.348,E2 -29554.348} C_VEL
LIN {X 0,Y 56.206,Z 309.823,A -85,B 0,C 180,E1 -29561.39,E2 -29561.39} C_VEL
LIN {X 0,Y 51.703,Z 312.193,A -85,B 0,C 180,E1 -29567.184,E2 -29567.184} C_VEL
LIN {X 0,Y 47.795,Z 313.997,A -85,B 0,C 180,E1 -29573.972,E2 -29573.972} C_VEL
LIN {X 0,Y 42.607,Z 316.463,A -85,B 0,C 180,E1 -29590.737,E2 -29590.737} C_VEL
LIN {X 0,Y 41.457,Z 317.063,A -85,B 0,C 180,E1 -29600.24,E2 -29600.24} C_VEL
LIN {X 0,Y 41.287,Z 317.227,A -85,B 0,C 180,E1 -29610,E2 -29610} C_VEL
LIN {X 0,Y 41.418,Z 317.062,A -85,B 0,C 180,E1 -29619.769,E2 -29619.769} C_VEL
LIN {X 0,Y 42.595,Z 316.462,A -85,B 0,C 180,E1 -29629.268,E2 -29629.268} C_VEL
LIN {X 0,Y 47.795,Z 313.997,A -85,B 0,C 180,E1 -29646.028,E2 -29646.028} C_VEL
LIN {X 0,Y 53.888,Z 311.041,A -85,B 0,C 180,E1 -29655.832,E2 -29655.832} C_VEL
LIN {X 0,Y 61.188,Z 307.051,A -85,B 0,C 180,E1 -29663.514,E2 -29663.514} C_VEL
LIN {X 0,Y 69.447,Z 301.832,A -85,B 0,C 180,E1 -29669.599,E2 -29669.599} C_VEL
LIN {X 0,Y 76.522,Z 296.657,A -85,B 0,C 180,E1 -29673.568,E2 -29673.568} C_VEL
LIN {X 0,Y 84.078,Z 290.343,A -85,B 0,C 180,E1 -29676.849,E2 -29676.849} C_VEL
LIN {X 0,Y 90.304,Z 284.397,A -85,B 0,C 180,E1 -29679.053,E2 -29679.053} C_VEL
LIN {X 0,Y 96.647,Z 277.475,A -85,B 0,C 180,E1 -29680.968,E2 -29680.968} C_VEL
LIN {X 0,Y 103.107,Z 269.304,A -85,B 0,C 180,E1 -29682.605,E2 -29682.605} C_VEL
LIN {X 0,Y 108.827,Z 260.799,A -85,B 0,C 180,E1 -29683.867,E2 -29683.867} C_VEL
LIN {X 0,Y 113.782,Z 252.092,A -85,B 0,C 180,E1 -29684.82,E2 -29684.82} C_VEL
LIN {X 0,Y 118.224,Z 242.638,A -85,B 0,C 180,E1 -29685.607,E2 -29685.607} C_VEL
LIN {X 0,Y 121.849,Z 232.987,A -85,B 0,C 180,E1 -29686.236,E2 -29686.236} C_VEL
LIN {X 0,Y 124.622,Z 223.453,A -85,B 0,C 180,E1 -29686.691,E2 -29686.691} C_VEL
LIN {X 0,Y 126.708,Z 213.255,A -85,B 0,C 180,E1 -29687.106,E2 -29687.106} C_VEL
LIN {X 0,Y 125.654,Z 209.535,A -85,B 0,C 180,E1 -29690.948,E2 -29690.948} C_VEL
LIN {X 0,Y 125.095,Z 207.482,A -85,B 0,C 180,E1 -29693.952,E2 -29693.952} C_VEL
LIN {X 0,Y 124.74,Z 204.564,A -85,B 0,C 180,E1 -29699.998,E2 -29699.998} C_VEL
LIN {X 0,Y 125.305,Z 208.302,A -85,B 0,C 180,E1 -29707.856,E2 -29707.856} C_VEL
LIN {X 0,Y 126.398,Z 212.268,A -85,B 0,C 180,E1 -29712.441,E2 -29712.441} C_VEL
LIN {X 0,Y 127.49,Z 217.154,A -85,B 0,C 180,E1 -29716.203,E2 -29716.203} C_VEL
LIN {X 0,Y 128.413,Z 223.827,A -85,B 0,C 180,E1 -29719.969,E2 -29719.969} C_VEL
LIN {X 0,Y 128.574,Z 229.597,A -85,B 0,C 180,E1 -29722.495,E2 -29722.495} C_VEL
LIN {X 0,Y 128.165,Z 237.665,A -85,B 0,C 180,E1 -29725.484,E2 -29725.484} C_VEL
LIN {X 0,Y 127.501,Z 247.037,A -85,B 0,C 180,E1 -29729.286,E2 -29729.286} C_VEL
LIN {X 0,Y 126.99,Z 256.213,A -85,B 0,C 180,E1 -29733.6,E2 -29733.6} C_VEL
LIN {X 0,Y 126.961,Z 263.413,A -85,B 0,C 180,E1 -29737.509,E2 -29737.509} C_VEL
LIN {X 0,Y 127.671,Z 271.91,A -85,B 0,C 180,E1 -29742.878,E2 -29742.878} C_VEL
LIN {X 0,Y 129.293,Z 279.234,A -85,B 0,C 180,E1 -29748.192,E2 -29748.192} C_VEL
LIN {X 0,Y 131.875,Z 285.123,A -85,B 0,C 180,E1 -29753.069,E2 -29753.069} C_VEL
LIN {X 0,Y 136.474,Z 291.454,A -85,B 0,C 180,E1 -29759.005,E2 -29759.005} C_VEL
LIN {X 0,Y 141.295,Z 295.847,A -85,B 0,C 180,E1 -29763.546,E2 -29763.546} C_VEL
LIN {X 0,Y 147.63,Z 299.906,A -85,B 0,C 180,E1 -29768.241,E2 -29768.241} C_VEL
LIN {X 0,Y 150.081,Z 301.602,A -85,B 0,C 180,E1 -29770.219,E2 -29770.219} C_VEL
LIN {X 0,Y 153.038,Z 304.57,A -85,B 0,C 180,E1 -29773.632,E2 -29773.632} C_VEL
LIN {X 0,Y 156.629,Z 306.991,A -85,B 0,C 180,E1 -29776.91,E2 -29776.91} C_VEL
LIN {X 0,Y 159.964,Z 307.898,A -85,B 0,C 180,E1 -29778.623,E2 -29778.623} C_VEL
LIN {X 0,Y 176.603,Z 310.177,A -85,B 0,C 180,E1 -29784.189,E2 -29784.189} C_VEL
LIN {X 0,Y 190.494,Z 310.876,A -85,B 0,C 180,E1 -29787.886,E2 -29787.886} C_VEL
LIN {X 0,Y 198.857,Z 310.823,A -85,B 0,C 180,E1 -29790,E2 -29790} C_VEL
LIN {X 0,Y 189.899,Z 310.86,A -85,B 0,C 180,E1 -29792.258,E2 -29792.258} C_VEL
LIN {X 0,Y 176.599,Z 310.184,A -85,B 0,C 180,E1 -29795.798,E2 -29795.798} C_VEL
LIN {X 0,Y 163.954,Z 308.647,A -85,B 0,C 180,E1 -29799.873,E2 -29799.873} C_VEL
LIN {X 0,Y 152.492,Z 306.183,A -85,B 0,C 180,E1 -29804.576,E2 -29804.576} C_VEL
LIN {X 0,Y 142.175,Z 302.502,A -85,B 0,C 180,E1 -29810.244,E2 -29810.244} C_VEL
LIN {X 0,Y 135.878,Z 299.023,A -85,B 0,C 180,E1 -29814.916,E2 -29814.916} C_VEL
LIN {X 0,Y 130.276,Z 294.515,A -85,B 0,C 180,E1 -29820.331,E2 -29820.331} C_VEL
LIN {X 0,Y 125.439,Z 288.149,A -85,B 0,C 180,E1 -29827.027,E2 -29827.027} C_VEL
LIN {X 0,Y 123.152,Z 282.696,A -85,B 0,C 180,E1 -29832.111,E2 -29832.111} C_VEL
LIN {X 0,Y 121.857,Z 276.109,A -85,B 0,C 180,E1 -29837.479,E2 -29837.479} C_VEL
LIN {X 0,Y 121.561,Z 267.148,A -85,B 0,C 180,E1 -29843.663,E2 -29843.663} C_VEL
LIN {X 0,Y 122.169,Z 258.32,A -85,B 0,C 180,E1 -29848.821,E2 -29848.821} C_VEL
LIN {X 0,Y 123.169,Z 250.197,A -85,B 0,C 180,E1 -29852.842,E2 -29852.842} C_VEL
LIN {X 0,Y 124.344,Z 241.247,A -85,B 0,C 180,E1 -29856.696,E2 -29856.696} C_VEL
LIN {X 0,Y 125.271,Z 233.898,A -85,B 0,C 180,E1 -29859.544,E2 -29859.544} C_VEL
LIN {X 0,Y 125.372,Z 227.893,A -85,B 0,C 180,E1 -29862.359,E2 -29862.359} C_VEL
LIN {X 0,Y 125.025,Z 222.428,A -85,B 0,C 180,E1 -29865.661,E2 -29865.661} C_VEL
LIN {X 0,Y 124.475,Z 218.388,A -85,B 0,C 180,E1 -29869.017,E2 -29869.017} C_VEL
LIN {X 0,Y 124.055,Z 215.808,A -85,B 0,C 180,E1 -29872.064,E2 -29872.064} C_VEL
LIN {X 0,Y 123.794,Z 214.273,A -85,B 0,C 180,E1 -29874.3,E2 -29874.3} C_VEL
LIN {X 0,Y 123.67,Z 211.8,A -85,B 0,C 180,E1 -29880.002,E2 -29880.002} C_VEL
LIN {X 0,Y 123.983,Z 214.95,A -85,B 0,C 180,E1 -29886.511,E2 -29886.511} C_VEL
LIN {X 0,Y 124.516,Z 217.683,A -85,B 0,C 180,E1 -29889.863,E2 -29889.863} C_VEL
LIN {X 0,Y 121.448,Z 229.497,A -85,B 0,C 180,E1 -29890.34,E2 -29890.34} C_VEL
LIN {X 0,Y 117.66,Z 240.091,A -85,B 0,C 180,E1 -29890.887,E2 -29890.887} C_VEL
LIN {X 0,Y 113.816,Z 248.639,A -85,B 0,C 180,E1 -29891.404,E2 -29891.404} C_VEL
LIN {X 0,Y 108.756,Z 257.909,A -85,B 0,C 180,E1 -29892.205,E2 -29892.205} C_VEL
LIN {X 0,Y 102.884,Z 266.846,A -85,B 0,C 180,E1 -29893.241,E2 -29893.241} C_VEL
LIN {X 0,Y 96.22,Z 275.367,A -85,B 0,C 180,E1 -29894.583,E2 -29894.583} C_VEL
LIN {X 0,Y 89.637,Z 282.58,A -85,B 0,C 180,E1 -29896.166,E2 -29896.166} C_VEL
LIN {X 0,Y 83.133,Z 288.776,A -85,B 0,C 180,E1 -29897.999,E2 -29897.999} C_VEL
LIN {X 0,Y 75.174,Z 295.309,A -85,B 0,C 180,E1 -29900.789,E2 -29900.789} C_VEL
LIN {X 0,Y 67.059,Z 301.033,A -85,B 0,C 180,E1 -29904.522,E2 -29904.522} C_VEL
LIN {X 0,Y 60.104,Z 305.306,A -85,B 0,C 180,E1 -29908.72,E2 -29908.72} C_VEL
LIN {X 0,Y 51.758,Z 309.631,A -85,B 0,C 180,E1 -29915.441,E2 -29915.441} C_VEL
LIN {X 0,Y 46.719,Z 312.002,A -85,B 0,C 180,E1 -29921.222,E2 -29921.222} C_VEL
LIN {X 0,Y 42.232,Z 313.805,A -85,B 0,C 180,E1 -29928.268,E2 -29928.268} C_VEL
LIN {X 0,Y 35.965,Z 316.272,A -85,B 0,C 180,E1 -29946.995,E2 -29946.995} C_VEL
LIN {X 0,Y 34.477,Z 316.872,A -85,B 0,C 180,E1 -29958.238,E2 -29958.238} C_VEL
LIN {X 0,Y 34.174,Z 317.036,A -85,B 0,C 180,E1 -29970,E2 -29970} C_VEL
LIN {X 0,Y 34.421,Z 316.871,A -85,B 0,C 180,E1 -29981.781,E2 -29981.781} C_VEL
LIN {X 0,Y 35.956,Z 316.272,A -85,B 0,C 180,E1 -29993.012,E2 -29993.012} C_VEL
LIN {X 0,Y 42.232,Z 313.805,A -85,B 0,C 180,E1 -30011.732,E2 -30011.732} C_VEL
LIN {X 0,Y 49.187,Z 310.85,A -85,B 0,C 180,E1 -30021.8,E2 -30021.8} C_VEL
LIN {X 0,Y 57.245,Z 306.86,A -85,B 0,C 180,E1 -30029.248,E2 -30029.248} C_VEL
LIN {X 0,Y 66.233,Z 301.566,A -85,B 0,C 180,E1 -30035.014,E2 -30035.014} C_VEL
LIN {X 0,Y 73.623,Z 296.466,A -85,B 0,C 180,E1 -30038.548,E2 -30038.548} C_VEL
LIN {X 0,Y 81.544,Z 290.152,A -85,B 0,C 180,E1 -30041.451,E2 -30041.451} C_VEL
LIN {X 0,Y 88.015,Z 284.206,A -85,B 0,C 180,E1 -30043.375,E2 -30043.375} C_VEL
LIN {X 0,Y 94.565,Z 277.284,A -85,B 0,C 180,E1 -30045.049,E2 -30045.049} C_VEL
LIN {X 0,Y 101.212,Z 269.113,A -85,B 0,C 180,E1 -30046.443,E2 -30046.443} C_VEL
LIN {X 0,Y 107.071,Z 260.609,A -85,B 0,C 180,E1 -30047.521,E2 -30047.521} C_VEL
LIN {X 0,Y 112.134,Z 251.901,A -85,B 0,C 180,E1 -30048.32,E2 -30048.32} C_VEL
LIN {X 0,Y 116.462,Z 242.925,A -85,B 0,C 180,E1 -30048.956,E2 -30048.956} C_VEL
LIN {X 0,Y 120.356,Z 232.796,A -85,B 0,C 180,E1 -30049.522,E2 -30049.522} C_VEL
LIN {X 0,Y 123.253,Z 222.99,A -85,B 0,C 180,E1 -30049.902,E2 -30049.902} C_VEL
LIN {X 0,Y 124.514,Z 217.691,A -85,B 0,C 180,E1 -30050.137,E2 -30050.137} C_VEL
LIN {X 0,Y 123.92,Z 214.643,A -85,B 0,C 180,E1 -30053.894,E2 -30053.894} C_VEL
LIN {X 0,Y 123.629,Z 211.79,A -85,B 0,C 180,E1 -30059.998,E2 -30059.998} C_VEL
LIN {X 0,Y 123.938,Z 214.983,A -85,B 0,C 180,E1 -30066.919,E2 -30066.919} C_VEL
LIN {X 0,Y 124.52,Z 218.539,A -85,B 0,C 180,E1 -30071.185,E2 -30071.185} C_VEL
LIN {X 0,Y 125.126,Z 223.35,A -85,B 0,C 180,E1 -30074.951,E2 -30074.951} C_VEL
LIN {X 0,Y 125.372,Z 227.893,A -85,B 0,C 180,E1 -30077.641,E2 -30077.641} C_VEL
LIN {X 0,Y 125.304,Z 232.947,A -85,B 0,C 180,E1 -30080.058,E2 -30080.058} C_VEL
LIN {X 0,Y 124.09,Z 243.603,A -85,B 0,C 180,E1 -30084.241,E2 -30084.241} C_VEL
LIN {X 0,Y 122.484,Z 255.4,A -85,B 0,C 180,E1 -30089.626,E2 -30089.626} C_VEL
LIN {X 0,Y 121.654,Z 264.429,A -85,B 0,C 180,E1 -30094.636,E2 -30094.636} C_VEL
LIN {X 0,Y 121.552,Z 271.899,A -85,B 0,C 180,E1 -30099.492,E2 -30099.492} C_VEL
LIN {X 0,Y 122.37,Z 279.489,A -85,B 0,C 180,E1 -30105.223,E2 -30105.223} C_VEL
LIN {X 0,Y 124.244,Z 285.626,A -85,B 0,C 180,E1 -30110.566,E2 -30110.566} C_VEL
LIN {X 0,Y 127.787,Z 291.73,A -85,B 0,C 180,E1 -30116.635,E2 -30116.635} C_VEL
LIN {X 0,Y 133.764,Z 297.541,A -85,B 0,C 180,E1 -30123.272,E2 -30123.272} C_VEL
LIN {X 0,Y 139.902,Z 301.415,A -85,B 0,C 180,E1 -30128.235,E2 -30128.235} C_VEL
LIN {X 0,Y 148.663,Z 305.013,A -85,B 0,C 180,E1 -30133.522,E2 -30133.522} C_VEL
LIN {X 0,Y 159.964,Z 307.898,A -85,B 0,C 180,E1 -30138.623,E2 -30138.623} C_VEL
LIN {X 0,Y 162.114,Z 308.571,A -85,B 0,C 180,E1 -30139.808,E2 -30139.808} C_VEL
LIN {X 0,Y 166.788,Z 310.596,A -85,B 0,C 180,E1 -30144.18,E2 -30144.18} C_VEL
LIN {X 0,Y 169.374,Z 310.862,A -85,B 0,C 180,E1 -30145.197,E2 -30145.197} C_VEL
LIN {X 0,Y 182.767,Z 311.223,A -85,B 0,C 180,E1 -30148.757,E2 -30148.757} C_VEL
LIN {X 0,Y 187.736,Z 311.116,A -85,B 0,C 180,E1 -30150,E2 -30150} C_VEL
LIN {X 0,Y 175.932,Z 311.105,A -85,B 0,C 180,E1 -30152.967,E2 -30152.967} C_VEL
LIN {X 0,Y 160.682,Z 310.076,A -85,B 0,C 180,E1 -30157.54,E2 -30157.54} C_VEL
LIN {X 0,Y 150.547,Z 308.605,A -85,B 0,C 180,E1 -30161.387,E2 -30161.387} C_VEL
LIN {X 0,Y 139.527,Z 305.832,A -85,B 0,C 180,E1 -30166.863,E2 -30166.863} C_VEL
LIN {X 0,Y 132.136,Z 302.785,A -85,B 0,C 180,E1 -30171.858,E2 -30171.858} C_VEL
LIN {X 0,Y 126.257,Z 299.215,A -85,B 0,C 180,E1 -30177.052,E2 -30177.052} C_VEL
LIN {X 0,Y 121.411,Z 294.612,A -85,B 0,C 180,E1 -30182.972,E2 -30182.972} C_VEL
LIN {X 0,Y 118.004,Z 289.047,A -85,B 0,C 180,E1 -30189.267,E2 -30189.267} C_VEL
LIN {X 0,Y 116.152,Z 282.271,A -85,B 0,C 180,E1 -30195.854,E2 -30195.854} C_VEL
LIN {X 0,Y 115.806,Z 274.72,A -85,B 0,C 180,E1 -30202.086,E2 -30202.086} C_VEL
LIN {X 0,Y 116.548,Z 266.801,A -85,B 0,C 180,E1 -30207.588,E2 -30207.588} C_VEL
LIN {X 0,Y 117.58,Z 260.433,A -85,B 0,C 180,E1 -30211.436,E2 -30211.436} C_VEL
LIN {X 0,Y 119.326,Z 251.302,A -85,B 0,C 180,E1 -30216.116,E2 -30216.116} C_VEL
LIN {X 0,Y 121.236,Z 241.809,A -85,B 0,C 180,E1 -30220.173,E2 -30220.173} C_VEL
LIN {X 0,Y 122.271,Z 235.453,A -85,B 0,C 180,E1 -30222.916,E2 -30222.916} C_VEL
LIN {X 0,Y 122.475,Z 230.154,A -85,B 0,C 180,E1 -30225.886,E2 -30225.886} C_VEL
LIN {X 0,Y 122.516,Z 226.654,A -85,B 0,C 180,E1 -30228.418,E2 -30228.418} C_VEL
LIN {X 0,Y 122.275,Z 223.043,A -85,B 0,C 180,E1 -30231.948,E2 -30231.948} C_VEL
LIN {X 0,Y 122.089,Z 220.978,A -85,B 0,C 180,E1 -30235.048,E2 -30235.048} C_VEL
LIN {X 0,Y 122.219,Z 218.931,A -85,B 0,C 180,E1 -30240.002,E2 -30240.002} C_VEL
LIN {X 0,Y 122.227,Z 221.695,A -85,B 0,C 180,E1 -30245.777,E2 -30245.777} C_VEL
LIN {X 0,Y 122.295,Z 222.409,A -85,B 0,C 180,E1 -30246.771,E2 -30246.771} C_VEL
LIN {X 0,Y 119.272,Z 232.609,A -85,B 0,C 180,E1 -30247.135,E2 -30247.135} C_VEL
LIN {X 0,Y 115.59,Z 242.081,A -85,B 0,C 180,E1 -30247.54,E2 -30247.54} C_VEL
LIN {X 0,Y 110.915,Z 251.711,A -85,B 0,C 180,E1 -30248.087,E2 -30248.087} C_VEL
LIN {X 0,Y 104.909,Z 261.769,A -85,B 0,C 180,E1 -30248.839,E2 -30248.839} C_VEL
LIN {X 0,Y 96.377,Z 273.259,A -85,B 0,C 180,E1 -30250.121,E2 -30250.121} C_VEL
LIN {X 0,Y 89.602,Z 280.763,A -85,B 0,C 180,E1 -30251.349,E2 -30251.349} C_VEL
LIN {X 0,Y 81.218,Z 288.585,A -85,B 0,C 180,E1 -30253.223,E2 -30253.223} C_VEL
LIN {X 0,Y 72.947,Z 295.118,A -85,B 0,C 180,E1 -30255.541,E2 -30255.541} C_VEL
LIN {X 0,Y 66.466,Z 299.62,A -85,B 0,C 180,E1 -30257.892,E2 -30257.892} C_VEL
LIN {X 0,Y 57.019,Z 305.114,A -85,B 0,C 180,E1 -30262.418,E2 -30262.418} C_VEL
LIN {X 0,Y 47.97,Z 309.44,A -85,B 0,C 180,E1 -30268.472,E2 -30268.472} C_VEL
LIN {X 0,Y 42.36,Z 311.81,A -85,B 0,C 180,E1 -30273.947,E2 -30273.947} C_VEL
LIN {X 0,Y 37.21,Z 313.614,A -85,B 0,C 180,E1 -30280.932,E2 -30280.932} C_VEL
LIN {X 0,Y 29.527,Z 316.08,A -85,B 0,C 180,E1 -30301.573,E2 -30301.573} C_VEL
LIN {X 0,Y 27.545,Z 316.681,A -85,B 0,C 180,E1 -30315.218,E2 -30315.218} C_VEL
LIN {X 0,Y 27.064,Z 316.845,A -85,B 0,C 180,E1 -30330,E2 -30330} C_VEL
LIN {X 0,Y 27.501,Z 316.68,A -85,B 0,C 180,E1 -30344.806,E2 -30344.806} C_VEL
LIN {X 0,Y 29.52,Z 316.08,A -85,B 0,C 180,E1 -30358.434,E2 -30358.434} C_VEL
LIN {X 0,Y 37.21,Z 313.614,A -85,B 0,C 180,E1 -30379.068,E2 -30379.068} C_VEL
LIN {X 0,Y 45.128,Z 310.659,A -85,B 0,C 180,E1 -30388.93,E2 -30388.93} C_VEL
LIN {X 0,Y 53.955,Z 306.669,A -85,B 0,C 180,E1 -30395.755,E2 -30395.755} C_VEL
LIN {X 0,Y 61.867,Z 302.397,A -85,B 0,C 180,E1 -30400.071,E2 -30400.071} C_VEL
LIN {X 0,Y 69.7,Z 297.43,A -85,B 0,C 180,E1 -30403.317,E2 -30403.317} C_VEL
LIN {X 0,Y 77.906,Z 291.337,A -85,B 0,C 180,E1 -30405.874,E2 -30405.874} C_VEL
LIN {X 0,Y 84.567,Z 285.64,A -85,B 0,C 180,E1 -30407.55,E2 -30407.55} C_VEL
LIN {X 0,Y 92.984,Z 277.093,A -85,B 0,C 180,E1 -30409.289,E2 -30409.289} C_VEL
LIN {X 0,Y 99.788,Z 268.923,A -85,B 0,C 180,E1 -30410.403,E2 -30410.403} C_VEL
LIN {X 0,Y 105.765,Z 260.418,A -85,B 0,C 180,E1 -30411.275,E2 -30411.275} C_VEL
LIN {X 0,Y 110.914,Z 251.711,A -85,B 0,C 180,E1 -30411.918,E2 -30411.918} C_VEL
LIN {X 0,Y 115.566,Z 242.13,A -85,B 0,C 180,E1 -30412.468,E2 -30412.468} C_VEL
LIN {X 0,Y 119.207,Z 232.788,A -85,B 0,C 180,E1 -30412.876,E2 -30412.876} C_VEL
LIN {X 0,Y 122.289,Z 222.421,A -85,B 0,C 180,E1 -30413.238,E2 -30413.238} C_VEL
LIN {X 0,Y 122.123,Z 220.806,A -85,B 0,C 180,E1 -30415.873,E2 -30415.873} C_VEL
LIN {X 0,Y 122.211,Z 218.95,A -85,B 0,C 180,E1 -30420.41,E2 -30420.41} C_VEL
LIN {X 0,Y 122.14,Z 221.551,A -85,B 0,C 180,E1 -30425.985,E2 -30425.985} C_VEL
LIN {X 0,Y 122.436,Z 224.774,A -85,B 0,C 180,E1 -30429.914,E2 -30429.914} C_VEL
LIN {X 0,Y 122.508,Z 228.848,A -85,B 0,C 180,E1 -30433.264,E2 -30433.264} C_VEL
LIN {X 0,Y 122.343,Z 234.652,A -85,B 0,C 180,E1 -30436.69,E2 -30436.69} C_VEL
LIN {X 0,Y 121.712,Z 239.044,A -85,B 0,C 180,E1 -30438.707,E2 -30438.707} C_VEL
LIN {X 0,Y 119.782,Z 249.018,A -85,B 0,C 180,E1 -30442.871,E2 -30442.871} C_VEL
LIN {X 0,Y 118.122,Z 257.21,A -85,B 0,C 180,E1 -30446.816,E2 -30446.816} C_VEL
LIN {X 0,Y 116.672,Z 265.647,A -85,B 0,C 180,E1 -30451.656,E2 -30451.656} C_VEL
LIN {X 0,Y 115.923,Z 272.461,A -85,B 0,C 180,E1 -30456.235,E2 -30456.235} C_VEL
LIN {X 0,Y 115.861,Z 279.644,A -85,B 0,C 180,E1 -30461.852,E2 -30461.852} C_VEL
LIN {X 0,Y 116.88,Z 285.895,A -85,B 0,C 180,E1 -30467.536,E2 -30467.536} C_VEL
LIN {X 0,Y 119.508,Z 292,A -85,B 0,C 180,E1 -30473.979,E2 -30473.979} C_VEL
LIN {X 0,Y 124.494,Z 297.762,A -85,B 0,C 180,E1 -30481.042,E2 -30481.042} C_VEL
LIN {X 0,Y 130.202,Z 301.743,A -85,B 0,C 180,E1 -30486.577,E2 -30486.577} C_VEL
LIN {X 0,Y 138.015,Z 305.306,A -85,B 0,C 180,E1 -30492.21,E2 -30492.21} C_VEL
LIN {X 0,Y 144.882,Z 307.405,A -85,B 0,C 180,E1 -30495.963,E2 -30495.963} C_VEL
LIN {X 0,Y 156.552,Z 309.613,A -85,B 0,C 180,E1 -30500.97,E2 -30500.97} C_VEL
LIN {X 0,Y 169.374,Z 310.862,A -85,B 0,C 180,E1 -30505.197,E2 -30505.197} C_VEL
LIN {X 0,Y 170.863,Z 311.001,A -85,B 0,C 180,E1 -30505.886,E2 -30505.886} C_VEL
LIN {X 0,Y 171.519,Z 311.255,A -85,B 0,C 180,E1 -30507.03,E2 -30507.03} C_VEL
LIN {X 0,Y 170.844,Z 311.538,A -85,B 0,C 180,E1 -30508.585,E2 -30508.585} C_VEL
LIN {X 0,Y 169.466,Z 311.597,A -85,B 0,C 180,E1 -30509.787,E2 -30509.787} C_VEL
LIN {X 0,Y 166.014,Z 311.643,A -85,B 0,C 180,E1 -30511.798,E2 -30511.798} C_VEL
LIN {X 0,Y 161.812,Z 311.396,A -85,B 0,C 180,E1 -30513.673,E2 -30513.673} C_VEL
LIN {X 0,Y 158.576,Z 311.223,A -85,B 0,C 180,E1 -30514.811,E2 -30514.811} C_VEL
LIN {X 0,Y 143.009,Z 309.625,A -85,B 0,C 180,E1 -30520.627,E2 -30520.627} C_VEL
LIN {X 0,Y 131.897,Z 307.092,A -85,B 0,C 180,E1 -30526.448,E2 -30526.448} C_VEL
LIN {X 0,Y 122.323,Z 303.069,A -85,B 0,C 180,E1 -30533.714,E2 -30533.714} C_VEL
LIN {X 0,Y 116.638,Z 299.007,A -85,B 0,C 180,E1 -30540.03,E2 -30540.03} C_VEL
LIN {X 0,Y 112.953,Z 294.667,A -85,B 0,C 180,E1 -30546.018,E2 -30546.018} C_VEL
LIN {X 0,Y 110.498,Z 288.808,A -85,B 0,C 180,E1 -30552.999,E2 -30552.999} C_VEL
LIN {X 0,Y 109.806,Z 282.94,A -85,B 0,C 180,E1 -30559.007,E2 -30559.007} C_VEL
LIN {X 0,Y 110.329,Z 275.982,A -85,B 0,C 180,E1 -30565.022,E2 -30565.022} C_VEL
LIN {X 0,Y 112.024,Z 267.04,A -85,B 0,C 180,E1 -30571.439,E2 -30571.439} C_VEL
LIN {X 0,Y 113.837,Z 260.028,A -85,B 0,C 180,E1 -30575.63,E2 -30575.63} C_VEL
LIN {X 0,Y 116.181,Z 251.401,A -85,B 0,C 180,E1 -30580.006,E2 -30580.006} C_VEL
LIN {X 0,Y 118.66,Z 241.874,A -85,B 0,C 180,E1 -30584.104,E2 -30584.104} C_VEL
LIN {X 0,Y 119.435,Z 237.51,A -85,B 0,C 180,E1 -30586.388,E2 -30586.388} C_VEL
LIN {X 0,Y 119.868,Z 233.682,A -85,B 0,C 180,E1 -30588.923,E2 -30588.923} C_VEL
LIN {X 0,Y 119.998,Z 230.696,A -85,B 0,C 180,E1 -30591.582,E2 -30591.582} C_VEL
LIN {X 0,Y 120.072,Z 228.592,A -85,B 0,C 180,E1 -30594.288,E2 -30594.288} C_VEL
LIN {X 0,Y 120.183,Z 227.253,A -85,B 0,C 180,E1 -30596.649,E2 -30596.649} C_VEL
LIN {X 0,Y 120.448,Z 225.94,A -85,B 0,C 180,E1 -30600.002,E2 -30600.002} C_VEL
LIN {X 0,Y 120.248,Z 227.442,A -85,B 0,C 180,E1 -30603.352,E2 -30603.352} C_VEL
LIN {X 0,Y 119.717,Z 229.116,A -85,B 0,C 180,E1 -30603.641,E2 -30603.641} C_VEL
LIN {X 0,Y 116.121,Z 239.023,A -85,B 0,C 180,E1 -30603.965,E2 -30603.965} C_VEL
LIN {X 0,Y 111.876,Z 248.257,A -85,B 0,C 180,E1 -30604.248,E2 -30604.248} C_VEL
LIN {X 0,Y 106.662,Z 257.528,A -85,B 0,C 180,E1 -30604.732,E2 -30604.732} C_VEL
LIN {X 0,Y 100.586,Z 266.466,A -85,B 0,C 180,E1 -30605.343,E2 -30605.343} C_VEL
LIN {X 0,Y 93.659,Z 274.986,A -85,B 0,C 180,E1 -30606.146,E2 -30606.146} C_VEL
LIN {X 0,Y 86.757,Z 282.198,A -85,B 0,C 180,E1 -30607.094,E2 -30607.094} C_VEL
LIN {X 0,Y 79.893,Z 288.395,A -85,B 0,C 180,E1 -30608.259,E2 -30608.259} C_VEL
LIN {X 0,Y 71.367,Z 294.926,A -85,B 0,C 180,E1 -30610.013,E2 -30610.013} C_VEL
LIN {X 0,Y 64.631,Z 299.428,A -85,B 0,C 180,E1 -30611.86,E2 -30611.86} C_VEL
LIN {X 0,Y 54.697,Z 304.923,A -85,B 0,C 180,E1 -30615.491,E2 -30615.491} C_VEL
LIN {X 0,Y 45.006,Z 309.248,A -85,B 0,C 180,E1 -30620.455,E2 -30620.455} C_VEL
LIN {X 0,Y 38.833,Z 311.619,A -85,B 0,C 180,E1 -30625.191,E2 -30625.191} C_VEL
LIN {X 0,Y 32.979,Z 313.422,A -85,B 0,C 180,E1 -30631.525,E2 -30631.525} C_VEL
LIN {X 0,Y 23.506,Z 315.889,A -85,B 0,C 180,E1 -30653.276,E2 -30653.276} C_VEL
LIN {X 0,Y 20.751,Z 316.491,A -85,B 0,C 180,E1 -30670.203,E2 -30670.203} C_VEL
LIN {X 0,Y 19.969,Z 316.655,A -85,B 0,C 180,E1 -30690,E2 -30690} C_VEL
LIN {X 0,Y 20.694,Z 316.489,A -85,B 0,C 180,E1 -30709.853,E2 -30709.853} C_VEL
LIN {X 0,Y 23.501,Z 315.889,A -85,B 0,C 180,E1 -30726.734,E2 -30726.734} C_VEL
LIN {X 0,Y 32.979,Z 313.422,A -85,B 0,C 180,E1 -30748.475,E2 -30748.475} C_VEL
LIN {X 0,Y 41.897,Z 310.467,A -85,B 0,C 180,E1 -30757.309,E2 -30757.309} C_VEL
LIN {X 0,Y 51.443,Z 306.478,A -85,B 0,C 180,E1 -30763.002,E2 -30763.002} C_VEL
LIN {X 0,Y 60.97,Z 301.537,A -85,B 0,C 180,E1 -30766.915,E2 -30766.915} C_VEL
LIN {X 0,Y 69.683,Z 296.083,A -85,B 0,C 180,E1 -30769.529,E2 -30769.529} C_VEL
LIN {X 0,Y 78.185,Z 289.77,A -85,B 0,C 180,E1 -30771.409,E2 -30771.409} C_VEL
LIN {X 0,Y 85.045,Z 283.825,A -85,B 0,C 180,E1 -30772.594,E2 -30772.594} C_VEL
LIN {X 0,Y 91.928,Z 276.902,A -85,B 0,C 180,E1 -30773.647,E2 -30773.647} C_VEL
LIN {X 0,Y 98.851,Z 268.732,A -85,B 0,C 180,E1 -30774.475,E2 -30774.475} C_VEL
LIN {X 0,Y 104.924,Z 260.228,A -85,B 0,C 180,E1 -30775.103,E2 -30775.103} C_VEL
LIN {X 0,Y 110.14,Z 251.52,A -85,B 0,C 180,E1 -30775.578,E2 -30775.578} C_VEL
LIN {X 0,Y 114.838,Z 241.97,A -85,B 0,C 180,E1 -30775.979,E2 -30775.979} C_VEL
LIN {X 0,Y 118.377,Z 233.068,A -85,B 0,C 180,E1 -30776.275,E2 -30776.275} C_VEL
LIN {X 0,Y 119.714,Z 229.115,A -85,B 0,C 180,E1 -30776.385,E2 -30776.385} C_VEL
LIN {X 0,Y 120.247,Z 227.446,A -85,B 0,C 180,E1 -30776.648,E2 -30776.648} C_VEL
LIN {X 0,Y 120.439,Z 225.971,A -85,B 0,C 180,E1 -30779.998,E2 -30779.998} C_VEL
LIN {X 0,Y 120.08,Z 228.589,A -85,B 0,C 180,E1 -30785.751,E2 -30785.751} C_VEL
LIN {X 0,Y 120.003,Z 230.682,A -85,B 0,C 180,E1 -30788.417,E2 -30788.417} C_VEL
LIN {X 0,Y 119.866,Z 233.681,A -85,B 0,C 180,E1 -30791.07,E2 -30791.07} C_VEL
